C03652=1111.482,258.279,-73.038,-178.384,10.028,149.558
C03653=1111.486,258.031,-73.009,-178.387,10.025,149.558
C03654=1111.491,257.782,-72.980,-178.389,10.023,149.558
C03655=1111.494,257.534,-72.951,-178.392,10.020,149.558
C03656=1111.499,257.286,-72.923,-178.395,10.017,149.558
C03657=1111.503,257.038,-72.894,-178.398,10.014,149.558
C03658=1111.507,256.790,-72.864,-178.401,10.011,149.558
C03659=1111.511,256.541,-72.836,-178.404,10.009,149.558
C03660=1111.516,256.293,-72.807,-178.406,10.006,149.558
C03661=1111.520,256.045,-72.778,-178.409,10.003,149.558
C03662=1111.524,255.832,-72.754,-178.410,10.001,149.558
C03663=1111.527,255.619,-72.729,-178.412,9.999,149.558
C03664=1111.531,255.406,-72.704,-178.414,9.998,149.558
C03665=1111.535,255.194,-72.680,-178.416,9.995,149.558
C03666=1111.538,254.981,-72.655,-178.418,9.993,149.558
C03667=1111.542,254.768,-72.630,-178.419,9.992,149.558
C03668=1111.545,254.555,-72.606,-178.422,9.990,149.559
C03669=1111.550,254.343,-72.581,-178.424,9.988,149.559
C03670=1111.554,254.094,-72.552,-178.426,9.986,149.559
C03671=1111.558,253.846,-72.524,-178.429,9.983,149.559
C03672=1111.562,253.598,-72.495,-178.431,9.981,149.559
C03673=1111.567,253.349,-72.466,-178.433,9.979,149.559
C03674=1111.571,253.101,-72.438,-178.436,9.976,149.559
C03675=1111.575,252.853,-72.408,-178.439,9.974,149.559
C03676=1111.579,252.605,-72.380,-178.442,9.971,149.559
C03677=1111.584,252.356,-72.352,-178.445,9.969,149.559
C03678=1111.587,252.108,-72.323,-178.447,9.967,149.560
C03679=1111.592,251.860,-72.294,-178.450,9.964,149.560
C03680=1111.597,251.611,-72.266,-178.453,9.962,149.560
C03681=1111.600,251.363,-72.237,-178.457,9.959,149.560
C03682=1111.605,251.115,-72.209,-178.460,9.956,149.560
C03683=1111.609,250.866,-72.180,-178.462,9.954,149.561
C03684=1111.614,250.618,-72.152,-178.466,9.951,149.561
C03685=1111.617,250.370,-72.123,-178.469,9.948,149.561
C03686=1111.622,250.121,-72.094,-178.472,9.946,149.561
C03687=1111.626,249.873,-72.067,-178.475,9.943,149.561
C03688=1111.631,249.624,-72.038,-178.479,9.940,149.562
C03689=1111.634,249.376,-72.010,-178.482,9.937,149.562
C03690=1111.640,249.128,-71.981,-178.485,9.935,149.562
C03691=1111.643,248.880,-71.953,-178.489,9.931,149.562
C03692=1111.647,248.632,-71.925,-178.492,9.928,149.562
C03693=1111.652,248.383,-71.896,-178.495,9.925,149.562
C03694=1111.656,248.134,-71.868,-178.499,9.922,149.563
C03695=1111.661,247.886,-71.839,-178.503,9.918,149.563
C03696=1111.664,247.637,-71.811,-178.506,9.915,149.563
C03697=1111.670,247.389,-71.783,-178.509,9.911,149.563
C03698=1111.673,247.141,-71.755,-178.511,9.908,149.563
C03699=1111.678,246.893,-71.727,-178.514,9.906,149.563
C03700=1111.682,246.644,-71.698,-178.516,9.903,149.563
C03701=1111.686,246.396,-71.671,-178.518,9.901,149.563
C03702=1111.690,246.147,-71.642,-178.520,9.898,149.562
C03703=1111.695,245.899,-71.614,-178.523,9.895,149.562
C03704=1111.699,245.651,-71.586,-178.525,9.892,149.562
C03705=1111.703,245.402,-71.558,-178.528,9.890,149.562
C03706=1111.708,245.154,-71.529,-178.530,9.887,149.562
C03707=1111.712,244.905,-71.501,-178.532,9.884,149.562
C03708=1111.716,244.657,-71.473,-178.535,9.882,149.562
C03709=1111.720,244.409,-71.445,-178.537,9.879,149.562
C03710=1111.725,244.161,-71.417,-178.539,9.877,149.562
C03711=1111.729,243.912,-71.390,-178.542,9.874,149.562
C03712=1111.733,243.664,-71.362,-178.544,9.872,149.562
C03713=1111.738,243.415,-71.333,-178.547,9.869,149.562
C03714=1111.742,243.167,-71.305,-178.549,9.867,149.562
C03715=1111.746,242.919,-71.277,-178.552,9.864,149.563
C03716=1111.750,242.670,-71.249,-178.554,9.861,149.562
C03717=1111.756,242.422,-71.222,-178.556,9.859,149.563
C03718=1111.759,242.209,-71.197,-178.558,9.856,149.563
C03719=1111.762,241.996,-71.174,-178.561,9.854,149.563
C03720=1111.766,241.783,-71.149,-178.563,9.852,149.563
C03721=1111.769,241.570,-71.126,-178.565,9.850,149.563
C03722=1111.774,241.357,-71.102,-178.567,9.847,149.563
C03723=1111.777,241.144,-71.078,-178.570,9.845,149.563
C03724=1111.781,240.931,-71.054,-178.572,9.843,149.563
C03725=1111.785,240.718,-71.030,-178.574,9.841,149.563
C03726=1111.789,240.470,-71.003,-178.576,9.839,149.563
C03727=1111.793,240.222,-70.975,-178.579,9.836,149.563
C03728=1111.797,239.974,-70.947,-178.582,9.833,149.563
C03729=1111.802,239.724,-70.919,-178.584,9.831,149.563
C03730=1111.806,239.477,-70.891,-178.587,9.828,149.563
C03731=1111.811,239.228,-70.864,-178.589,9.826,149.563
C03732=1111.815,238.980,-70.836,-178.592,9.823,149.563
C03733=1111.819,238.732,-70.808,-178.595,9.820,149.564
C03734=1111.823,238.482,-70.781,-178.597,9.818,149.563
C03735=1111.827,238.235,-70.753,-178.600,9.815,149.564
C03736=1111.832,237.987,-70.725,-178.603,9.812,149.564
C03737=1111.836,237.738,-70.698,-178.605,9.811,149.564
C03738=1111.841,237.489,-70.669,-178.608,9.808,149.564
C03739=1111.846,237.241,-70.642,-178.610,9.805,149.564
C03740=1111.849,236.992,-70.614,-178.613,9.803,149.564
C03741=1111.854,236.744,-70.587,-178.616,9.800,149.564
C03742=1111.858,236.496,-70.559,-178.618,9.797,149.564
C03743=1111.862,236.247,-70.532,-178.621,9.794,149.564
C03744=1111.867,235.999,-70.504,-178.623,9.792,149.564
C03745=1111.871,235.750,-70.477,-178.626,9.789,149.564
C03746=1111.875,235.502,-70.449,-178.629,9.787,149.565
C03747=1111.880,235.253,-70.422,-178.632,9.784,149.565
C03748=1111.884,235.005,-70.395,-178.634,9.782,149.565
C03749=1111.888,234.756,-70.367,-178.637,9.779,149.565
C03750=1111.893,234.508,-70.339,-178.640,9.776,149.565
C03751=1111.897,234.260,-70.312,-178.643,9.773,149.565
C03752=1111.901,234.011,-70.284,-178.646,9.771,149.565
C03753=1111.906,233.762,-70.257,-178.648,9.767,149.565
C03754=1111.910,233.514,-70.229,-178.651,9.765,149.565
C03755=1111.915,233.266,-70.202,-178.654,9.763,149.565
C03756=1111.918,233.017,-70.176,-178.657,9.760,149.565
C03757=1111.923,232.769,-70.148,-178.660,9.757,149.566
C03758=1111.927,232.520,-70.121,-178.662,9.754,149.566
C03759=1111.932,232.272,-70.094,-178.665,9.751,149.566
C03760=1111.936,232.023,-70.065,-178.668,9.749,149.566
C03761=1111.940,231.775,-70.038,-178.670,9.745,149.566
C03762=1111.945,231.526,-70.011,-178.673,9.743,149.566
C03763=1111.950,231.278,-69.984,-178.676,9.740,149.566
C03764=1111.953,231.029,-69.956,-178.679,9.737,149.566
C03765=1111.957,230.781,-69.930,-178.682,9.734,149.566
C03766=1111.962,230.533,-69.903,-178.685,9.731,149.566
C03767=1111.967,230.284,-69.876,-178.687,9.728,149.566
C03768=1111.971,230.035,-69.848,-178.690,9.726,149.566
C03769=1111.975,229.786,-69.821,-178.693,9.723,149.566
C03770=1111.980,229.539,-69.793,-178.696,9.720,149.566
C03771=1111.984,229.290,-69.767,-178.699,9.717,149.566
C03772=1111.988,229.042,-69.740,-178.701,9.714,149.566
C03773=1111.993,228.793,-69.713,-178.704,9.711,149.566
C03774=1111.997,228.580,-69.689,-178.707,9.708,149.566
C03775=1112.001,228.367,-69.666,-178.709,9.706,149.566
C03776=1112.004,228.154,-69.644,-178.711,9.704,149.566
C03777=1112.007,227.941,-69.620,-178.713,9.701,149.566
C03778=1112.011,227.728,-69.596,-178.716,9.699,149.566
C03779=1112.015,227.514,-69.574,-178.718,9.695,149.566
C03780=1112.019,227.302,-69.551,-178.720,9.693,149.566
C03781=1112.022,227.089,-69.528,-178.723,9.690,149.566
C03782=1112.027,226.841,-69.501,-178.726,9.687,149.566
C03783=1112.032,226.592,-69.474,-178.728,9.684,149.566
C03784=1112.035,226.343,-69.447,-178.731,9.681,149.566
C03785=1112.040,226.095,-69.420,-178.733,9.678,149.566
C03786=1112.044,225.846,-69.393,-178.736,9.675,149.566
C03787=1112.048,225.598,-69.366,-178.739,9.672,149.566
C03788=1112.053,225.349,-69.340,-178.741,9.669,149.566
C03789=1112.058,225.101,-69.313,-178.744,9.666,149.566
C03790=1112.062,224.853,-69.286,-178.746,9.663,149.566
C03791=1112.067,224.604,-69.259,-178.749,9.660,149.566
C03792=1112.070,224.356,-69.233,-178.751,9.657,149.566
C03793=1112.075,224.107,-69.206,-178.754,9.653,149.566
C03794=1112.079,223.858,-69.178,-178.756,9.650,149.566
C03795=1112.083,223.609,-69.152,-178.759,9.647,149.566
C03796=1112.088,223.361,-69.125,-178.761,9.644,149.566
C03797=1112.092,223.113,-69.099,-178.764,9.641,149.566
C03798=1112.097,222.864,-69.072,-178.766,9.638,149.566
C03799=1112.101,222.616,-69.045,-178.769,9.635,149.565
C03800=1112.106,222.367,-69.019,-178.771,9.632,149.565
C03801=1112.110,222.118,-68.992,-178.774,9.629,149.565
C03802=1112.114,221.870,-68.966,-178.777,9.625,149.565
C03803=1112.119,221.621,-68.939,-178.778,9.623,149.565
C03804=1112.123,221.373,-68.913,-178.781,9.620,149.565
C03805=1112.128,221.124,-68.886,-178.783,9.617,149.565
C03806=1112.132,220.876,-68.860,-178.786,9.614,149.565
C03807=1112.137,220.627,-68.833,-178.788,9.610,149.565
C03808=1112.140,220.379,-68.806,-178.791,9.607,149.565
C03809=1112.145,220.130,-68.780,-178.793,9.604,149.565
C03810=1112.149,219.882,-68.754,-178.796,9.601,149.565
C03811=1112.154,219.633,-68.727,-178.798,9.598,149.564
C03812=1112.158,219.384,-68.701,-178.800,9.595,149.564
C03813=1112.163,219.136,-68.674,-178.802,9.592,149.564
C03814=1112.167,218.887,-68.648,-178.805,9.589,149.564
C03815=1112.171,218.639,-68.621,-178.807,9.586,149.564
C03816=1112.176,218.390,-68.594,-178.810,9.583,149.564
C03817=1112.180,218.142,-68.569,-178.812,9.580,149.564
C03818=1112.185,217.893,-68.542,-178.814,9.577,149.564
C03819=1112.189,217.644,-68.516,-178.816,9.574,149.564
C03820=1112.193,217.396,-68.489,-178.819,9.571,149.564
C03821=1112.198,217.147,-68.463,-178.821,9.568,149.563
C03822=1112.202,216.899,-68.437,-178.823,9.565,149.563
C03823=1112.206,216.651,-68.411,-178.825,9.562,149.563
C03824=1112.211,216.402,-68.385,-178.828,9.559,149.563
C03825=1112.215,216.153,-68.358,-178.830,9.556,149.563
C03826=1112.219,215.905,-68.333,-178.832,9.553,149.563
C03827=1112.224,215.656,-68.306,-178.834,9.550,149.563
C03828=1112.228,215.407,-68.280,-178.837,9.547,149.563
C03829=1112.232,215.159,-68.253,-178.839,9.544,149.563
C03830=1112.237,214.946,-68.231,-178.840,9.542,149.562
C03831=1112.240,214.733,-68.209,-178.843,9.538,149.562
C03832=1112.244,214.519,-68.186,-178.845,9.536,149.562
C03833=1112.248,214.307,-68.164,-178.847,9.534,149.562
C03834=1112.251,214.093,-68.142,-178.848,9.531,149.562
C03835=1112.256,213.880,-68.119,-178.850,9.529,149.562
C03836=1112.259,213.667,-68.097,-178.852,9.526,149.562
C03837=1112.263,213.454,-68.074,-178.854,9.524,149.562
C03838=1112.267,213.205,-68.048,-178.856,9.521,149.562
C03839=1112.272,212.956,-68.022,-178.860,9.517,149.562
C03840=1112.276,212.708,-67.997,-178.862,9.514,149.562
C03841=1112.281,212.460,-67.970,-178.865,9.511,149.562
C03842=1112.285,212.211,-67.944,-178.868,9.508,149.562
C03843=1112.290,211.962,-67.918,-178.871,9.505,149.562
C03844=1112.294,211.713,-67.893,-178.874,9.501,149.562
C03845=1112.298,211.465,-67.866,-178.876,9.499,149.562
C03846=1112.303,211.217,-67.840,-178.879,9.496,149.562
C03847=1112.307,210.968,-67.814,-178.882,9.493,149.562
C03848=1112.312,210.719,-67.789,-178.885,9.489,149.562
C03849=1112.316,210.470,-67.763,-178.888,9.486,149.562
C03850=1112.320,210.221,-67.737,-178.891,9.483,149.562
C03851=1112.325,209.973,-67.712,-178.894,9.480,149.562
C03852=1112.330,209.725,-67.685,-178.896,9.478,149.562
C03853=1112.334,209.476,-67.659,-178.899,9.475,149.562
C03854=1112.338,209.227,-67.633,-178.903,9.471,149.562
C03855=1112.343,208.979,-67.608,-178.905,9.468,149.562
C03856=1112.347,208.730,-67.582,-178.908,9.465,149.562
C03857=1112.351,208.482,-67.556,-178.911,9.462,149.563
C03858=1112.356,208.233,-67.531,-178.914,9.459,149.562
C03859=1112.360,207.985,-67.505,-178.916,9.457,149.563
C03860=1112.365,207.736,-67.479,-178.919,9.454,149.563
C03861=1112.369,207.487,-67.454,-178.922,9.451,149.563
C03862=1112.373,207.238,-67.428,-178.925,9.448,149.563
C03863=1112.378,206.990,-67.403,-178.928,9.445,149.563
C03864=1112.382,206.741,-67.377,-178.931,9.442,149.563
C03865=1112.386,206.492,-67.351,-178.934,9.439,149.563
C03866=1112.391,206.244,-67.326,-178.937,9.436,149.563
C03867=1112.396,205.995,-67.301,-178.940,9.433,149.563
C03868=1112.400,205.746,-67.275,-178.943,9.430,149.563
C03869=1112.405,205.498,-67.249,-178.945,9.427,149.563
C03870=1112.409,205.249,-67.224,-178.948,9.425,149.564
C03871=1112.413,205.000,-67.198,-178.951,9.422,149.564
C03872=1112.418,204.752,-67.173,-178.954,9.419,149.564
C03873=1112.423,204.503,-67.148,-178.957,9.416,149.564
C03874=1112.427,204.254,-67.122,-178.960,9.413,149.564
C03875=1112.432,204.006,-67.096,-178.963,9.410,149.564
C03876=1112.436,203.757,-67.071,-178.966,9.408,149.564
C03877=1112.441,203.508,-67.046,-178.968,9.405,149.564
C03878=1112.445,203.260,-67.020,-178.971,9.402,149.564
C03879=1112.449,203.011,-66.995,-178.974,9.399,149.564
C03880=1112.454,202.763,-66.969,-178.976,9.396,149.564
C03881=1112.459,202.513,-66.944,-178.980,9.392,149.565
C03882=1112.462,202.265,-66.919,-178.983,9.390,149.565
C03883=1112.467,202.017,-66.894,-178.986,9.387,149.565
C03884=1112.472,201.767,-66.869,-178.988,9.384,149.565
C03885=1112.476,201.519,-66.843,-178.991,9.381,149.565
C03886=1112.480,201.305,-66.822,-178.993,9.379,149.565
C03887=1112.484,201.093,-66.800,-178.996,9.376,149.565
C03888=1112.488,200.879,-66.778,-178.998,9.374,149.565
C03889=1112.491,200.666,-66.757,-179.001,9.371,149.565
C03890=1112.496,200.453,-66.735,-179.003,9.369,149.565
C03891=1112.499,200.239,-66.713,-179.006,9.366,149.565
C03892=1112.503,200.026,-66.692,-179.008,9.364,149.565
C03893=1112.506,199.813,-66.670,-179.011,9.361,149.565
C03894=1112.512,199.564,-66.645,-179.013,9.358,149.565
C03895=1112.515,199.316,-66.620,-179.016,9.355,149.565
C03896=1112.520,199.067,-66.595,-179.019,9.352,149.565
C03897=1112.524,198.818,-66.570,-179.021,9.349,149.565
C03898=1112.530,198.569,-66.545,-179.024,9.346,149.565
C03899=1112.533,198.321,-66.520,-179.027,9.343,149.565
C03900=1112.538,198.072,-66.495,-179.029,9.340,149.565
C03901=1112.542,197.823,-66.469,-179.033,9.336,149.565
C03902=1112.547,197.575,-66.445,-179.035,9.333,149.565
C03903=1112.551,197.326,-66.420,-179.038,9.330,149.565
C03904=1112.556,197.077,-66.395,-179.041,9.327,149.565
C03905=1112.560,196.828,-66.370,-179.043,9.324,149.565
C03906=1112.565,196.580,-66.345,-179.046,9.321,149.565
C03907=1112.569,196.331,-66.320,-179.049,9.318,149.565
C03908=1112.574,196.082,-66.296,-179.051,9.315,149.565
C03909=1112.578,195.834,-66.270,-179.052,9.312,149.565
C03910=1112.582,195.585,-66.246,-179.055,9.309,149.565
C03911=1112.587,195.336,-66.221,-179.056,9.306,149.565
C03912=1112.592,195.087,-66.196,-179.059,9.303,149.565
C03913=1112.596,194.839,-66.172,-179.061,9.301,149.565
C03914=1112.601,194.590,-66.147,-179.063,9.297,149.564
C03915=1112.605,194.341,-66.123,-179.065,9.295,149.564
C03916=1112.609,194.093,-66.097,-179.067,9.292,149.564
C03917=1112.614,193.844,-66.072,-179.069,9.290,149.564
C03918=1112.619,193.595,-66.048,-179.071,9.287,149.564
C03919=1112.623,193.346,-66.023,-179.073,9.284,149.564
C03920=1112.627,193.098,-65.998,-179.075,9.282,149.564
C03921=1112.632,192.849,-65.973,-179.078,9.278,149.564
C03922=1112.636,192.600,-65.949,-179.080,9.276,149.564
C03923=1112.641,192.352,-65.924,-179.082,9.273,149.564
C03924=1112.645,192.103,-65.900,-179.085,9.270,149.564
C03925=1112.650,191.854,-65.875,-179.087,9.268,149.564
C03926=1112.654,191.605,-65.850,-179.089,9.264,149.563
C03927=1112.659,191.357,-65.826,-179.091,9.262,149.563
C03928=1112.663,191.108,-65.801,-179.093,9.259,149.563
C03929=1112.668,190.859,-65.776,-179.095,9.256,149.563
C03930=1112.672,190.610,-65.752,-179.097,9.253,149.563
C03931=1112.677,190.362,-65.728,-179.099,9.251,149.563
C03932=1112.681,190.113,-65.703,-179.102,9.248,149.563
C03933=1112.686,189.864,-65.679,-179.104,9.245,149.563
C03934=1112.691,189.615,-65.654,-179.106,9.242,149.563
C03935=1112.695,189.366,-65.629,-179.109,9.239,149.563
C03936=1112.700,189.118,-65.605,-179.111,9.237,149.563
C03937=1112.705,188.869,-65.581,-179.113,9.234,149.563
C03938=1112.709,188.620,-65.556,-179.115,9.231,149.563
C03939=1112.713,188.371,-65.532,-179.118,9.228,149.563
C03940=1112.718,188.123,-65.508,-179.120,9.225,149.563
C03941=1112.722,187.873,-65.483,-179.122,9.223,149.563
C03942=1112.726,187.660,-65.462,-179.124,9.221,149.563
C03943=1112.730,187.447,-65.441,-179.126,9.217,149.563
C03944=1112.734,187.234,-65.420,-179.128,9.215,149.563
C03945=1112.738,187.021,-65.399,-179.130,9.213,149.563
C03946=1112.742,186.807,-65.378,-179.132,9.210,149.563
C03947=1112.745,186.593,-65.358,-179.134,9.208,149.563
C03948=1112.750,186.380,-65.337,-179.136,9.206,149.563
C03949=1112.753,186.167,-65.316,-179.138,9.203,149.563
C03950=1112.758,185.918,-65.292,-179.140,9.200,149.562
C03951=1112.762,185.669,-65.267,-179.143,9.198,149.563
C03952=1112.766,185.421,-65.243,-179.146,9.194,149.563
C03953=1112.772,185.172,-65.218,-179.148,9.192,149.563
C03954=1112.776,184.923,-65.195,-179.150,9.189,149.563
C03955=1112.780,184.674,-65.171,-179.153,9.186,149.562
C03956=1112.785,184.425,-65.146,-179.155,9.184,149.562
C03957=1112.790,184.177,-65.122,-179.157,9.180,149.562
C03958=1112.794,183.928,-65.098,-179.160,9.177,149.562
C03959=1112.799,183.679,-65.074,-179.162,9.174,149.562
C03960=1112.803,183.430,-65.049,-179.165,9.171,149.562
C03961=1112.808,183.182,-65.025,-179.167,9.169,149.562
C03962=1112.812,182.933,-65.001,-179.169,9.166,149.562
C03963=1112.817,182.684,-64.978,-179.172,9.163,149.562
C03964=1112.820,182.435,-64.953,-179.174,9.160,149.562
C03965=1112.826,182.186,-64.929,-179.177,9.156,149.562
C03966=1112.830,181.937,-64.905,-179.179,9.153,149.562
C03967=1112.835,181.689,-64.881,-179.181,9.151,149.562
C03968=1112.839,181.440,-64.857,-179.184,9.148,149.562
C03969=1112.844,181.191,-64.834,-179.186,9.145,149.562
C03970=1112.848,180.942,-64.809,-179.189,9.142,149.562
C03971=1112.853,180.694,-64.785,-179.191,9.139,149.562
C03972=1112.857,180.445,-64.761,-179.194,9.135,149.562
C03973=1112.862,180.196,-64.737,-179.196,9.132,149.562
C03974=1112.866,179.947,-64.714,-179.199,9.129,149.562
C03975=1112.871,179.699,-64.690,-179.201,9.126,149.562
C03976=1112.876,179.450,-64.667,-179.204,9.123,149.562
C03977=1112.879,179.201,-64.642,-179.206,9.119,149.561
C03978=1112.884,178.952,-64.618,-179.208,9.117,149.561
C03979=1112.889,178.703,-64.594,-179.210,9.114,149.561
C03980=1112.894,178.454,-64.570,-179.212,9.111,149.561
C03981=1112.898,178.205,-64.547,-179.214,9.108,149.561
C03982=1112.903,177.957,-64.523,-179.217,9.105,149.561
C03983=1112.907,177.708,-64.499,-179.219,9.102,149.561
C03984=1112.912,177.459,-64.476,-179.221,9.099,149.561
C03985=1112.916,177.210,-64.452,-179.223,9.096,149.561
C03986=1112.921,176.961,-64.428,-179.225,9.093,149.560
C03987=1112.925,176.712,-64.404,-179.227,9.090,149.560
C03988=1112.930,176.463,-64.381,-179.230,9.087,149.560
C03989=1112.934,176.215,-64.357,-179.231,9.085,149.560
C03990=1112.939,175.966,-64.333,-179.234,9.081,149.560
C03991=1112.943,175.717,-64.310,-179.236,9.078,149.560
C03992=1112.948,175.468,-64.286,-179.238,9.076,149.560
C03993=1112.953,175.219,-64.262,-179.240,9.073,149.560
C03994=1112.957,174.970,-64.239,-179.243,9.069,149.560
C03995=1112.962,174.722,-64.215,-179.244,9.067,149.559
C03996=1112.966,174.473,-64.192,-179.247,9.064,149.559
C03997=1112.971,174.224,-64.168,-179.249,9.061,149.559
C03998=1112.975,174.011,-64.148,-179.251,9.058,149.559
C03999=1112.978,173.797,-64.128,-179.253,9.055,149.559
C04000=1112.983,173.583,-64.108,-179.255,9.053,149.559
C04001=1112.987,173.370,-64.088,-179.257,9.051,149.559
C04002=1112.990,173.157,-64.067,-179.259,9.047,149.559
C04003=1112.994,172.943,-64.047,-179.261,9.045,149.559
C04004=1112.998,172.730,-64.027,-179.262,9.043,149.559
C04005=1113.002,172.516,-64.007,-179.264,9.040,149.559
C04006=1113.007,172.268,-63.983,-179.266,9.037,149.558
C04007=1113.011,172.019,-63.960,-179.268,9.035,149.558
C04008=1113.016,171.770,-63.936,-179.271,9.031,149.558
C04009=1113.020,171.521,-63.914,-179.273,9.028,149.558
C04010=1113.025,171.272,-63.890,-179.275,9.026,149.558
C04011=1113.029,171.023,-63.866,-179.277,9.022,149.558
C04012=1113.034,170.774,-63.843,-179.279,9.019,149.558
C04013=1113.038,170.525,-63.820,-179.282,9.016,149.558
C04014=1113.043,170.276,-63.796,-179.284,9.014,149.558
C04015=1113.048,170.027,-63.773,-179.286,9.010,149.557
C04016=1113.052,169.778,-63.750,-179.288,9.007,149.557
C04017=1113.057,169.530,-63.727,-179.290,9.005,149.557
C04018=1113.062,169.281,-63.704,-179.292,9.001,149.557
C04019=1113.066,169.032,-63.680,-179.295,8.998,149.557
C04020=1113.071,168.783,-63.657,-179.297,8.995,149.557
C04021=1113.075,168.534,-63.634,-179.299,8.992,149.557
C04022=1113.080,168.285,-63.611,-179.301,8.989,149.557
C04023=1113.084,168.036,-63.588,-179.304,8.986,149.557
C04024=1113.089,167.787,-63.564,-179.305,8.983,149.557
C04025=1113.093,167.539,-63.541,-179.308,8.980,149.556
C04026=1113.098,167.289,-63.518,-179.310,8.977,149.556
C04027=1113.103,167.041,-63.495,-179.313,8.974,149.556
C04028=1113.108,166.792,-63.472,-179.314,8.971,149.556
C04029=1113.112,166.543,-63.449,-179.317,8.968,149.556
C04030=1113.117,166.294,-63.426,-179.319,8.965,149.556
C04031=1113.121,166.045,-63.402,-179.322,8.962,149.556
C04032=1113.125,165.797,-63.379,-179.323,8.959,149.556
C04033=1113.130,165.548,-63.356,-179.326,8.956,149.556
C04034=1113.135,165.299,-63.333,-179.328,8.952,149.555
C04035=1113.139,165.051,-63.310,-179.330,8.949,149.555
C04036=1113.144,164.802,-63.287,-179.333,8.946,149.555
C04037=1113.149,164.552,-63.264,-179.334,8.943,149.555
C04038=1113.153,164.303,-63.242,-179.337,8.940,149.555
C04039=1113.158,164.054,-63.218,-179.339,8.937,149.555
C04040=1113.163,163.806,-63.195,-179.341,8.934,149.555
C04041=1113.167,163.557,-63.172,-179.343,8.931,149.555
C04042=1113.172,163.307,-63.150,-179.345,8.928,149.554
C04043=1113.176,163.059,-63.127,-179.348,8.925,149.554
C04044=1113.180,162.810,-63.104,-179.350,8.921,149.554
C04045=1113.185,162.562,-63.081,-179.352,8.918,149.554
C04046=1113.190,162.312,-63.059,-179.354,8.915,149.554
C04047=1113.195,162.063,-63.035,-179.356,8.912,149.554
C04048=1113.199,161.814,-63.013,-179.358,8.909,149.554
C04049=1113.203,161.565,-62.989,-179.361,8.906,149.554
C04050=1113.208,161.317,-62.967,-179.363,8.902,149.553
C04051=1113.213,161.068,-62.944,-179.366,8.899,149.553
C04052=1113.217,160.819,-62.921,-179.367,8.896,149.553
C04053=1113.222,160.569,-62.899,-179.370,8.893,149.553
C04054=1113.226,160.356,-62.879,-179.372,8.890,149.553
C04055=1113.230,160.143,-62.859,-179.373,8.887,149.553
C04056=1113.234,159.929,-62.840,-179.375,8.885,149.553
C04057=1113.237,159.715,-62.821,-179.377,8.882,149.553
C04058=1113.241,159.502,-62.801,-179.379,8.879,149.553
C04059=1113.246,159.288,-62.783,-179.381,8.877,149.552
C04060=1113.249,159.075,-62.763,-179.383,8.874,149.552
C04061=1113.253,158.861,-62.743,-179.385,8.871,149.552
C04062=1113.258,158.611,-62.720,-179.387,8.868,149.552
C04063=1113.263,158.363,-62.698,-179.389,8.864,149.552
C04064=1113.267,158.114,-62.676,-179.391,8.861,149.552
C04065=1113.272,157.865,-62.653,-179.393,8.858,149.551
C04066=1113.277,157.616,-62.631,-179.395,8.855,149.551
C04067=1113.281,157.367,-62.608,-179.398,8.852,149.551
C04068=1113.286,157.118,-62.586,-179.400,8.848,149.551
C04069=1113.290,156.870,-62.563,-179.402,8.845,149.551
C04070=1113.295,156.620,-62.540,-179.405,8.842,149.551
C04071=1113.299,156.372,-62.518,-179.407,8.838,149.550
C04072=1113.305,156.123,-62.495,-179.409,8.835,149.550
C04073=1113.309,155.874,-62.473,-179.411,8.832,149.550
C04074=1113.313,155.625,-62.451,-179.413,8.828,149.550
C04075=1113.319,155.376,-62.428,-179.415,8.825,149.550
C04076=1113.323,155.127,-62.406,-179.417,8.822,149.550
C04077=1113.327,154.878,-62.384,-179.419,8.819,149.549
C04078=1113.332,154.629,-62.361,-179.422,8.815,149.549
C04079=1113.336,154.380,-62.339,-179.424,8.812,149.549
C04080=1113.341,154.131,-62.317,-179.426,8.809,149.549
C04081=1113.346,153.882,-62.293,-179.428,8.805,149.549
C04082=1113.350,153.633,-62.271,-179.430,8.802,149.548
C04083=1113.355,153.384,-62.250,-179.433,8.799,149.548
C04084=1113.359,153.135,-62.228,-179.435,8.795,149.548
C04085=1113.365,152.887,-62.205,-179.437,8.792,149.548
C04086=1113.369,152.637,-62.183,-179.439,8.788,149.548
C04087=1113.373,152.388,-62.161,-179.441,8.785,149.547
C04088=1113.378,152.139,-62.139,-179.444,8.782,149.547
C04089=1113.383,151.890,-62.116,-179.446,8.778,149.547
C04090=1113.388,151.642,-62.094,-179.448,8.775,149.547
C04091=1113.392,151.392,-62.072,-179.450,8.771,149.547
C04092=1113.397,151.144,-62.050,-179.452,8.768,149.546
C04093=1113.402,150.894,-62.027,-179.454,8.764,149.546
C04094=1113.406,150.646,-62.005,-179.456,8.761,149.546
C04095=1113.411,150.397,-61.983,-179.458,8.757,149.546
C04096=1113.415,150.148,-61.961,-179.461,8.753,149.546
C04097=1113.420,149.899,-61.939,-179.463,8.750,149.546
C04098=1113.425,149.650,-61.918,-179.466,8.746,149.545
C04099=1113.430,149.400,-61.895,-179.468,8.743,149.545
C04100=1113.434,149.152,-61.873,-179.470,8.739,149.545
C04101=1113.439,148.902,-61.851,-179.472,8.736,149.545
C04102=1113.444,148.654,-61.830,-179.474,8.732,149.544
C04103=1113.448,148.404,-61.808,-179.476,8.729,149.544
C04104=1113.453,148.156,-61.786,-179.478,8.725,149.544
C04105=1113.457,147.906,-61.764,-179.480,8.722,149.544
C04106=1113.462,147.658,-61.741,-179.482,8.718,149.543
C04107=1113.467,147.409,-61.719,-179.485,8.714,149.543
C04108=1113.472,147.160,-61.698,-179.487,8.711,149.543
C04109=1113.476,146.910,-61.676,-179.489,8.707,149.542
C04110=1113.480,146.698,-61.657,-179.490,8.704,149.542
C04111=1113.484,146.483,-61.638,-179.493,8.701,149.542
C04112=1113.488,146.270,-61.620,-179.495,8.697,149.542
C04113=1113.492,146.056,-61.601,-179.496,8.695,149.542
C04114=1113.496,145.842,-61.582,-179.498,8.691,149.542
C04115=1113.500,145.629,-61.563,-179.500,8.689,149.541
C04116=1113.504,145.415,-61.544,-179.502,8.685,149.541
C04117=1113.508,145.201,-61.526,-179.504,8.682,149.541
C04118=1113.512,144.952,-61.504,-179.505,8.678,149.540
C04119=1113.517,144.703,-61.482,-179.506,8.675,149.540
C04120=1113.522,144.455,-61.461,-179.509,8.671,149.540
C04121=1113.526,144.205,-61.439,-179.510,8.668,149.539
C04122=1113.531,143.956,-61.418,-179.512,8.665,149.539
C04123=1113.536,143.707,-61.396,-179.513,8.661,149.539
C04124=1113.540,143.458,-61.374,-179.515,8.658,149.538
C04125=1113.545,143.210,-61.352,-179.516,8.654,149.538
C04126=1113.550,142.960,-61.330,-179.518,8.651,149.538
C04127=1113.555,142.711,-61.309,-179.519,8.648,149.537
C04128=1113.559,142.462,-61.287,-179.522,8.644,149.537
C04129=1113.564,142.213,-61.266,-179.523,8.641,149.537
C04130=1113.568,141.965,-61.245,-179.525,8.637,149.536
C04131=1113.573,141.715,-61.223,-179.527,8.634,149.536
C04132=1113.577,141.466,-61.201,-179.528,8.631,149.536
C04133=1113.582,141.217,-61.180,-179.530,8.627,149.535
C04134=1113.587,140.967,-61.158,-179.531,8.624,149.535
C04135=1113.592,140.719,-61.137,-179.533,8.621,149.535
C04136=1113.597,140.470,-61.115,-179.535,8.617,149.534
C04137=1113.601,140.221,-61.093,-179.537,8.613,149.534
C04138=1113.605,139.972,-61.073,-179.538,8.611,149.534
C04139=1113.610,139.723,-61.051,-179.540,8.607,149.533
C04140=1113.615,139.473,-61.030,-179.542,8.603,149.533
C04141=1113.620,139.225,-61.008,-179.543,8.600,149.533
C04142=1113.624,138.976,-60.986,-179.545,8.597,149.533
C04143=1113.629,138.726,-60.965,-179.547,8.593,149.532
C04144=1113.633,138.478,-60.944,-179.548,8.590,149.532
C04145=1113.638,138.228,-60.923,-179.550,8.587,149.532
C04146=1113.643,137.979,-60.901,-179.552,8.583,149.531
C04147=1113.647,137.730,-60.879,-179.553,8.580,149.531
C04148=1113.652,137.482,-60.859,-179.555,8.577,149.531
C04149=1113.657,137.233,-60.837,-179.557,8.573,149.530
C04150=1113.661,136.983,-60.816,-179.558,8.570,149.530
C04151=1113.666,136.734,-60.794,-179.560,8.567,149.530
C04152=1113.671,136.485,-60.774,-179.562,8.563,149.529
C04153=1113.676,136.237,-60.752,-179.563,8.560,149.529
C04154=1113.680,135.987,-60.731,-179.565,8.556,149.529
C04155=1113.685,135.738,-60.709,-179.567,8.553,149.529
C04156=1113.689,135.489,-60.689,-179.569,8.550,149.528
C04157=1113.694,135.241,-60.667,-179.571,8.546,149.528
C04158=1113.699,134.991,-60.646,-179.572,8.543,149.528
C04159=1113.704,134.741,-60.625,-179.574,8.540,149.527
C04160=1113.708,134.493,-60.604,-179.576,8.536,149.527
C04161=1113.713,134.244,-60.583,-179.577,8.533,149.527
C04162=1113.718,133.995,-60.561,-179.579,8.530,149.526
C04163=1113.722,133.745,-60.540,-179.581,8.526,149.526
C04164=1113.727,133.496,-60.519,-179.582,8.524,149.526
C04165=1113.732,133.248,-60.498,-179.584,8.520,149.526
C04166=1113.736,133.034,-60.480,-179.585,8.517,149.525
C04167=1113.740,132.820,-60.462,-179.587,8.514,149.525
C04168=1113.744,132.606,-60.444,-179.589,8.511,149.525
C04169=1113.747,132.392,-60.426,-179.590,8.508,149.525
C04170=1113.752,132.179,-60.407,-179.592,8.505,149.524
C04171=1113.756,131.965,-60.390,-179.593,8.503,149.524
C04172=1113.760,131.751,-60.371,-179.595,8.500,149.524
C04173=1113.764,131.537,-60.354,-179.596,8.497,149.524
C04174=1113.769,131.288,-60.333,-179.598,8.493,149.523
C04175=1113.774,131.039,-60.311,-179.600,8.490,149.523
C04176=1113.778,130.790,-60.291,-179.601,8.487,149.523
C04177=1113.783,130.540,-60.269,-179.603,8.483,149.522
C04178=1113.787,130.292,-60.249,-179.605,8.480,149.522
C04179=1113.792,130.043,-60.227,-179.606,8.477,149.522
C04180=1113.797,129.794,-60.207,-179.608,8.474,149.522
C04181=1113.802,129.545,-60.186,-179.610,8.470,149.521
C04182=1113.807,129.295,-60.165,-179.612,8.467,149.521
C04183=1113.811,129.046,-60.145,-179.614,8.463,149.521
C04184=1113.816,128.798,-60.123,-179.616,8.460,149.521
C04185=1113.821,128.549,-60.103,-179.617,8.457,149.520
C04186=1113.825,128.299,-60.081,-179.619,8.453,149.520
C04187=1113.830,128.050,-60.061,-179.621,8.450,149.520
C04188=1113.835,127.801,-60.040,-179.622,8.447,149.520
C04189=1113.839,127.552,-60.020,-179.624,8.443,149.519
C04190=1113.845,127.302,-59.999,-179.626,8.440,149.519
C04191=1113.849,127.054,-59.978,-179.627,8.437,149.519
C04192=1113.854,126.804,-59.957,-179.629,8.434,149.518
C04193=1113.858,126.556,-59.936,-179.631,8.430,149.518
C04194=1113.863,126.307,-59.916,-179.633,8.427,149.518
C04195=1113.868,126.058,-59.895,-179.635,8.423,149.518
C04196=1113.872,125.809,-59.874,-179.637,8.420,149.517
C04197=1113.877,125.560,-59.853,-179.638,8.417,149.517
C04198=1113.882,125.311,-59.833,-179.640,8.413,149.517
C04199=1113.886,125.061,-59.812,-179.642,8.410,149.516
C04200=1113.891,124.812,-59.791,-179.643,8.407,149.516
C04201=1113.895,124.563,-59.771,-179.645,8.403,149.516
C04202=1113.901,124.313,-59.750,-179.647,8.400,149.515
C04203=1113.905,124.065,-59.730,-179.649,8.396,149.515
C04204=1113.909,123.816,-59.709,-179.650,8.394,149.515
C04205=1113.915,123.566,-59.688,-179.652,8.390,149.515
C04206=1113.919,123.317,-59.669,-179.654,8.386,149.514
C04207=1113.924,123.068,-59.648,-179.656,8.383,149.514
C04208=1113.929,122.819,-59.627,-179.658,8.380,149.514
C04209=1113.933,122.570,-59.607,-179.660,8.376,149.514
C04210=1113.938,122.321,-59.587,-179.661,8.373,149.513
C04211=1113.943,122.071,-59.566,-179.663,8.370,149.513
C04212=1113.947,121.822,-59.545,-179.665,8.366,149.513
C04213=1113.952,121.573,-59.525,-179.667,8.363,149.513
C04214=1113.957,121.324,-59.505,-179.668,8.360,149.512
C04215=1113.962,121.075,-59.484,-179.670,8.356,149.512
C04216=1113.966,120.826,-59.464,-179.672,8.353,149.512
C04217=1113.972,120.577,-59.443,-179.673,8.350,149.511
C04218=1113.976,120.328,-59.423,-179.675,8.346,149.511
C04219=1113.981,120.079,-59.403,-179.677,8.343,149.511
C04220=1113.986,119.830,-59.383,-179.679,8.339,149.511
C04221=1113.991,119.580,-59.362,-179.681,8.336,149.510
C04222=1113.994,119.367,-59.345,-179.682,8.334,149.510
C04223=1113.998,119.152,-59.327,-179.684,8.330,149.510
C04224=1114.002,118.939,-59.310,-179.685,8.327,149.509
C04225=1114.006,118.725,-59.293,-179.687,8.324,149.509
C04226=1114.011,118.511,-59.275,-179.688,8.322,149.509
C04227=1114.015,118.297,-59.258,-179.689,8.319,149.509
C04228=1114.019,118.084,-59.240,-179.691,8.316,149.509
C04229=1114.023,117.869,-59.223,-179.693,8.313,149.508
C04230=1114.027,117.620,-59.202,-179.695,8.309,149.508
C04231=1114.033,117.371,-59.183,-179.696,8.307,149.508
C04232=1114.037,117.122,-59.162,-179.698,8.303,149.507
C04233=1114.042,116.873,-59.142,-179.700,8.299,149.507
C04234=1114.046,116.624,-59.122,-179.702,8.296,149.507
C04235=1114.051,116.374,-59.102,-179.703,8.293,149.507
C04236=1114.056,116.125,-59.082,-179.705,8.289,149.506
C04237=1114.061,115.876,-59.061,-179.707,8.286,149.506
C04238=1114.065,115.627,-59.041,-179.709,8.282,149.506
C04239=1114.070,115.378,-59.022,-179.710,8.279,149.505
C04240=1114.075,115.129,-59.001,-179.712,8.276,149.505
C04241=1114.080,114.880,-58.982,-179.714,8.272,149.505
C04242=1114.085,114.630,-58.961,-179.716,8.268,149.505
C04243=1114.089,114.381,-58.941,-179.718,8.265,149.504
C04244=1114.094,114.132,-58.921,-179.720,8.262,149.504
C04245=1114.099,113.883,-58.901,-179.722,8.258,149.504
C04246=1114.104,113.634,-58.881,-179.723,8.255,149.503
C04247=1114.108,113.384,-58.861,-179.725,8.251,149.503
C04248=1114.113,113.136,-58.841,-179.727,8.248,149.503
C04249=1114.118,112.886,-58.821,-179.728,8.244,149.503
C04250=1114.123,112.638,-58.801,-179.730,8.241,149.502
C04251=1114.127,112.388,-58.782,-179.732,8.237,149.502
C04252=1114.132,112.139,-58.761,-179.734,8.234,149.502
C04253=1114.137,111.890,-58.742,-179.736,8.231,149.501
C04254=1114.142,111.641,-58.722,-179.738,8.227,149.501
C04255=1114.146,111.392,-58.702,-179.739,8.223,149.501
C04256=1114.151,111.142,-58.682,-179.741,8.220,149.501
C04257=1114.156,110.893,-58.663,-179.743,8.216,149.500
C04258=1114.161,110.644,-58.643,-179.745,8.213,149.500
C04259=1114.166,110.395,-58.623,-179.747,8.209,149.500
C04260=1114.170,110.146,-58.603,-179.749,8.206,149.499
C04261=1114.175,109.896,-58.583,-179.751,8.202,149.499
C04262=1114.180,109.647,-58.564,-179.754,8.198,149.499
C04263=1114.185,109.398,-58.544,-179.756,8.194,149.499
C04264=1114.189,109.149,-58.524,-179.758,8.191,149.499
C04265=1114.194,108.899,-58.504,-179.760,8.187,149.498
C04266=1114.199,108.651,-58.485,-179.762,8.183,149.498
C04267=1114.204,108.401,-58.465,-179.764,8.180,149.498
C04268=1114.208,108.152,-58.445,-179.766,8.176,149.497
C04269=1114.213,107.903,-58.426,-179.768,8.172,149.497
C04270=1114.218,107.654,-58.406,-179.770,8.168,149.497
C04271=1114.223,107.404,-58.387,-179.772,8.165,149.497
C04272=1114.227,107.155,-58.366,-179.774,8.161,149.496
C04273=1114.232,106.906,-58.347,-179.776,8.157,149.496
C04274=1114.237,106.657,-58.327,-179.777,8.153,149.495
C04275=1114.241,106.408,-58.308,-179.779,8.150,149.495
C04276=1114.247,106.159,-58.289,-179.782,8.146,149.495
C04277=1114.251,105.909,-58.269,-179.784,8.142,149.495
C04278=1114.256,105.695,-58.252,-179.785,8.139,149.494
C04279=1114.259,105.481,-58.236,-179.787,8.136,149.494
C04280=1114.264,105.268,-58.219,-179.788,8.132,149.494
C04281=1114.267,105.053,-58.202,-179.790,8.129,149.494
C04282=1114.272,104.839,-58.186,-179.792,8.126,149.493
C04283=1114.276,104.626,-58.169,-179.793,8.122,149.493
C04284=1114.280,104.411,-58.152,-179.795,8.120,149.493
C04285=1114.284,104.198,-58.135,-179.797,8.116,149.492
C04286=1114.289,103.949,-58.116,-179.798,8.112,149.492
C04287=1114.294,103.699,-58.096,-179.800,8.109,149.492
C04288=1114.299,103.450,-58.077,-179.802,8.105,149.491
C04289=1114.303,103.201,-58.058,-179.804,8.101,149.491
C04290=1114.308,102.952,-58.038,-179.806,8.097,149.491
C04291=1114.313,102.703,-58.019,-179.807,8.094,149.490
C04292=1114.317,102.453,-58.001,-179.809,8.090,149.490
C04293=1114.323,102.204,-57.982,-179.811,8.086,149.490
C04294=1114.328,101.954,-57.962,-179.812,8.082,149.489
C04295=1114.332,101.706,-57.943,-179.815,8.079,149.489
C04296=1114.337,101.456,-57.924,-179.816,8.075,149.488
C04297=1114.342,101.207,-57.904,-179.818,8.071,149.488
C04298=1114.346,100.958,-57.885,-179.819,8.067,149.488
C04299=1114.351,100.709,-57.866,-179.821,8.064,149.487
C04300=1114.356,100.460,-57.846,-179.823,8.060,149.487
C04301=1114.360,100.210,-57.827,-179.825,8.056,149.487
C04302=1114.366,99.961,-57.809,-179.826,8.052,149.486
C04303=1114.371,99.711,-57.789,-179.828,8.048,149.486
C04304=1114.375,99.463,-57.770,-179.830,8.045,149.485
C04305=1114.380,99.213,-57.751,-179.831,8.041,149.485
C04306=1114.385,98.965,-57.732,-179.833,8.037,149.485
C04307=1114.390,98.714,-57.713,-179.835,8.033,149.484
C04308=1114.395,98.466,-57.694,-179.836,8.029,149.484
C04309=1114.399,98.216,-57.675,-179.838,8.025,149.483
C04310=1114.404,97.968,-57.655,-179.840,8.022,149.483
C04311=1114.409,97.718,-57.637,-179.842,8.018,149.483
C04312=1114.414,97.469,-57.618,-179.843,8.014,149.482
C04313=1114.418,97.220,-57.599,-179.845,8.010,149.482
C04314=1114.423,96.971,-57.579,-179.846,8.006,149.481
C04315=1114.428,96.721,-57.561,-179.848,8.002,149.481
C04316=1114.433,96.472,-57.542,-179.850,7.998,149.480
C04317=1114.437,96.223,-57.523,-179.851,7.994,149.480
C04318=1114.443,95.973,-57.504,-179.853,7.991,149.480
C04319=1114.447,95.725,-57.485,-179.854,7.987,149.479
C04320=1114.452,95.474,-57.466,-179.856,7.983,149.479
C04321=1114.457,95.226,-57.448,-179.858,7.979,149.478
C04322=1114.462,94.976,-57.428,-179.859,7.975,149.478
C04323=1114.467,94.727,-57.410,-179.860,7.972,149.477
C04324=1114.471,94.478,-57.390,-179.862,7.968,149.477
C04325=1114.476,94.228,-57.372,-179.863,7.964,149.477
C04326=1114.482,93.979,-57.353,-179.865,7.960,149.476
C04327=1114.486,93.730,-57.334,-179.867,7.956,149.476
C04328=1114.491,93.481,-57.316,-179.868,7.952,149.475
C04329=1114.495,93.231,-57.296,-179.869,7.948,149.475
C04330=1114.500,92.982,-57.278,-179.871,7.944,149.474
C04331=1114.506,92.733,-57.259,-179.872,7.941,149.474
C04332=1114.510,92.484,-57.241,-179.873,7.937,149.473
C04333=1114.514,92.235,-57.222,-179.875,7.933,149.473
C04334=1114.519,92.021,-57.205,-179.876,7.930,149.472
C04335=1114.523,91.806,-57.190,-179.878,7.926,149.472
C04336=1114.528,91.592,-57.174,-179.879,7.923,149.472
C04337=1114.531,91.378,-57.158,-179.880,7.920,149.471
C04338=1114.535,91.164,-57.142,-179.882,7.917,149.471
C04339=1114.540,90.950,-57.125,-179.883,7.914,149.470
C04340=1114.544,90.736,-57.110,-179.884,7.910,149.470
C04341=1114.548,90.522,-57.094,-179.884,7.907,149.470
C04342=1114.553,90.273,-57.076,-179.886,7.903,149.469
C04343=1114.558,90.023,-57.057,-179.887,7.899,149.469
C04344=1114.563,89.774,-57.038,-179.889,7.895,149.468
C04345=1114.567,89.525,-57.020,-179.890,7.891,149.468
C04346=1114.572,89.275,-57.002,-179.891,7.888,149.467
C04347=1114.577,89.027,-56.982,-179.893,7.884,149.467
C04348=1114.582,88.777,-56.964,-179.894,7.880,149.466
C04349=1114.586,88.527,-56.946,-179.896,7.876,149.466
C04350=1114.592,88.279,-56.927,-179.896,7.873,149.465
C04351=1114.597,88.029,-56.909,-179.898,7.869,149.465
C04352=1114.601,87.780,-56.890,-179.899,7.865,149.464
C04353=1114.606,87.531,-56.872,-179.901,7.861,149.464
C04354=1114.611,87.282,-56.853,-179.902,7.858,149.463
C04355=1114.616,87.032,-56.835,-179.903,7.854,149.463
C04356=1114.620,86.782,-56.817,-179.904,7.849,149.462
C04357=1114.625,86.534,-56.798,-179.906,7.845,149.462
C04358=1114.630,86.285,-56.780,-179.907,7.842,149.461
C04359=1114.636,86.035,-56.762,-179.908,7.838,149.461
C04360=1114.640,85.785,-56.743,-179.910,7.834,149.460
C04361=1114.645,85.537,-56.725,-179.910,7.831,149.460
C04362=1114.649,85.288,-56.707,-179.912,7.827,149.459
C04363=1114.654,85.038,-56.689,-179.913,7.823,149.459
C04364=1114.659,84.788,-56.670,-179.914,7.819,149.458
C04365=1114.664,84.539,-56.652,-179.915,7.815,149.458
C04366=1114.669,84.290,-56.634,-179.917,7.812,149.457
C04367=1114.674,84.041,-56.615,-179.917,7.808,149.456
C04368=1114.678,83.792,-56.597,-179.919,7.804,149.456
C04369=1114.683,83.542,-56.579,-179.920,7.800,149.455
C04370=1114.689,83.293,-56.560,-179.921,7.797,149.455
C04371=1114.694,83.044,-56.542,-179.922,7.793,149.454
C04372=1114.699,82.795,-56.524,-179.923,7.789,149.454
C04373=1114.703,82.545,-56.506,-179.924,7.785,149.453
C04374=1114.708,82.295,-56.488,-179.926,7.781,149.453
C04375=1114.713,82.046,-56.470,-179.926,7.778,149.452
C04376=1114.717,81.798,-56.451,-179.928,7.774,149.452
C04377=1114.722,81.549,-56.433,-179.929,7.770,149.451
C04378=1114.727,81.299,-56.415,-179.930,7.766,149.451
C04379=1114.731,81.049,-56.397,-179.931,7.763,149.450
C04380=1114.736,80.800,-56.379,-179.932,7.759,149.450
C04381=1114.742,80.551,-56.360,-179.933,7.755,149.449
C04382=1114.747,80.302,-56.342,-179.934,7.752,149.448
C04383=1114.752,80.052,-56.324,-179.935,7.747,149.448
C04384=1114.757,79.803,-56.306,-179.936,7.744,149.447
C04385=1114.761,79.553,-56.288,-179.937,7.740,149.447
C04386=1114.766,79.304,-56.270,-179.938,7.737,149.446
C04387=1114.771,79.055,-56.252,-179.940,7.733,149.446
C04388=1114.776,78.806,-56.234,-179.941,7.729,149.445
C04389=1114.781,78.556,-56.217,-179.942,7.725,149.445
C04390=1114.785,78.342,-56.201,-179.943,7.722,149.444
C04391=1114.789,78.128,-56.186,-179.944,7.719,149.444
C04392=1114.793,77.914,-56.170,-179.944,7.715,149.443
C04393=1114.797,77.700,-56.155,-179.944,7.713,149.443
C04394=1114.801,77.485,-56.140,-179.945,7.710,149.442
C04395=1114.805,77.271,-56.124,-179.946,7.707,149.442
C04396=1114.810,77.057,-56.109,-179.947,7.704,149.441
C04397=1114.814,76.843,-56.093,-179.948,7.700,149.441
C04398=1114.819,76.593,-56.075,-179.949,7.696,149.440
C04399=1114.824,76.344,-56.057,-179.951,7.693,149.440
C04400=1114.829,76.095,-56.039,-179.953,7.689,149.439
C04401=1114.834,75.846,-56.021,-179.954,7.684,149.439
C04402=1114.839,75.596,-56.004,-179.955,7.680,149.438
C04403=1114.843,75.347,-55.987,-179.957,7.677,149.438
C04404=1114.848,75.098,-55.969,-179.958,7.673,149.437
C04405=1114.853,74.849,-55.951,-179.960,7.668,149.437
C04406=1114.858,74.600,-55.933,-179.961,7.664,149.436
C04407=1114.863,74.350,-55.915,-179.963,7.661,149.436
C04408=1114.868,74.101,-55.897,-179.964,7.656,149.435
C04409=1114.872,73.851,-55.879,-179.965,7.652,149.435
C04410=1114.877,73.602,-55.861,-179.966,7.649,149.434
C04411=1114.882,73.352,-55.844,-179.968,7.645,149.434
C04412=1114.887,73.103,-55.827,-179.969,7.641,149.433
C04413=1114.892,72.854,-55.809,-179.971,7.637,149.433
C04414=1114.897,72.604,-55.791,-179.972,7.633,149.433
C04415=1114.902,72.355,-55.773,-179.974,7.629,149.432
C04416=1114.907,72.106,-55.755,-179.975,7.625,149.431
C04417=1114.911,71.857,-55.737,-179.976,7.621,149.431
C04418=1114.916,71.607,-55.721,-179.978,7.617,149.431
C04419=1114.921,71.358,-55.703,-179.979,7.613,149.430
C04420=1114.926,71.108,-55.685,-179.981,7.609,149.429
C04421=1114.931,70.859,-55.667,-179.982,7.605,149.429
C04422=1114.936,70.610,-55.649,-179.983,7.602,149.428
C04423=1114.940,70.360,-55.633,-179.984,7.598,149.428
C04424=1114.945,70.111,-55.615,-179.986,7.594,149.428
C04425=1114.951,69.862,-55.598,-179.987,7.590,149.427
C04426=1114.956,69.613,-55.580,-179.989,7.586,149.426
C04427=1114.961,69.363,-55.563,-179.990,7.582,149.426
C04428=1114.965,69.114,-55.545,-179.992,7.578,149.426
C04429=1114.970,68.865,-55.527,-179.993,7.574,149.425
C04430=1114.975,68.616,-55.511,-179.994,7.570,149.425
C04431=1114.980,68.366,-55.493,-179.996,7.566,149.424
C04432=1114.985,68.117,-55.475,-179.997,7.561,149.423
C04433=1114.990,67.867,-55.457,-179.998,7.558,149.423
C04434=1114.994,67.618,-55.441,-180.000,7.554,149.423
C04435=1115.000,67.368,-55.423,179.999,7.550,149.422
C04436=1115.004,67.119,-55.406,179.998,7.546,149.421
C04437=1115.009,66.869,-55.389,179.997,7.542,149.421
C04438=1115.014,66.620,-55.371,179.995,7.538,149.420
C04439=1115.020,66.371,-55.354,179.993,7.534,149.420
C04440=1115.024,66.122,-55.337,179.992,7.530,149.419
C04441=1115.029,65.872,-55.319,179.991,7.526,149.419
C04442=1115.034,65.623,-55.303,179.989,7.522,149.418
C04443=1115.038,65.374,-55.285,179.989,7.519,149.418
C04444=1115.044,65.124,-55.267,179.987,7.515,149.417
C04445=1115.048,64.875,-55.250,179.986,7.511,149.417
C04446=1115.053,64.661,-55.236,179.984,7.507,149.417
C04447=1115.056,64.446,-55.221,179.984,7.503,149.416
C04448=1115.061,64.232,-55.206,179.983,7.500,149.415
C04449=1115.066,64.018,-55.191,179.981,7.496,149.415
C04450=1115.069,63.804,-55.176,179.980,7.493,149.415
C04451=1115.074,63.590,-55.161,179.979,7.490,149.414
C04452=1115.078,63.375,-55.147,179.978,7.486,149.414
C04453=1115.082,63.161,-55.132,179.977,7.483,149.413
C04454=1115.087,62.911,-55.115,179.975,7.479,149.413
C04455=1115.092,62.662,-55.097,179.974,7.475,149.412
C04456=1115.097,62.413,-55.081,179.972,7.471,149.412
C04457=1115.102,62.163,-55.064,179.971,7.468,149.411
C04458=1115.106,61.914,-55.047,179.970,7.464,149.411
C04459=1115.111,61.665,-55.029,179.969,7.460,149.410
C04460=1115.116,61.415,-55.012,179.968,7.455,149.410
C04461=1115.122,61.166,-54.996,179.966,7.451,149.409
C04462=1115.126,60.917,-54.979,179.965,7.447,149.409
C04463=1115.131,60.667,-54.962,179.963,7.443,149.408
C04464=1115.136,60.418,-54.944,179.962,7.439,149.408
C04465=1115.141,60.168,-54.927,179.961,7.436,149.407
C04466=1115.146,59.919,-54.911,179.960,7.432,149.407
C04467=1115.151,59.670,-54.893,179.959,7.428,149.406
C04468=1115.156,59.420,-54.877,179.957,7.424,149.405
C04469=1115.161,59.170,-54.859,179.956,7.419,149.405
C04470=1115.166,58.922,-54.843,179.955,7.415,149.404
C04471=1115.170,58.672,-54.826,179.953,7.411,149.404
C04472=1115.176,58.422,-54.809,179.952,7.407,149.403
C04473=1115.180,58.173,-54.792,179.951,7.404,149.403
C04474=1115.186,57.924,-54.775,179.950,7.400,149.402
C04475=1115.190,57.675,-54.758,179.949,7.396,149.402
C04476=1115.194,57.425,-54.742,179.947,7.392,149.401
C04477=1115.200,57.176,-54.725,179.946,7.388,149.401
C04478=1115.205,56.927,-54.708,179.945,7.383,149.400
C04479=1115.210,56.677,-54.691,179.943,7.380,149.400
C04480=1115.214,56.427,-54.674,179.942,7.376,149.399
C04481=1115.220,56.179,-54.658,179.941,7.372,149.399
C04482=1115.225,55.929,-54.641,179.940,7.368,149.398
C04483=1115.229,55.679,-54.624,179.939,7.364,149.397
C04484=1115.234,55.431,-54.608,179.937,7.360,149.397
C04485=1115.240,55.181,-54.590,179.936,7.355,149.396
C04486=1115.244,54.931,-54.574,179.935,7.351,149.396
C04487=1115.249,54.682,-54.558,179.934,7.348,149.395
C04488=1115.255,54.432,-54.541,179.933,7.344,149.395
C04489=1115.259,54.183,-54.524,179.931,7.340,149.394
C04490=1115.264,53.934,-54.508,179.930,7.336,149.394
C04491=1115.269,53.684,-54.491,179.929,7.331,149.393
C04492=1115.274,53.435,-54.474,179.927,7.328,149.393
C04493=1115.279,53.186,-54.458,179.926,7.323,149.392
C04494=1115.283,52.936,-54.441,179.925,7.319,149.391
C04495=1115.290,52.687,-54.425,179.924,7.316,149.391
C04496=1115.294,52.437,-54.408,179.923,7.312,149.390
C04497=1115.299,52.188,-54.391,179.921,7.308,149.390
C04498=1115.304,51.939,-54.375,179.920,7.303,149.389
C04499=1115.309,51.689,-54.358,179.919,7.299,149.389
C04500=1115.314,51.440,-54.342,179.918,7.295,149.388
C04501=1115.319,51.190,-54.326,179.917,7.291,149.387
C04502=1115.323,50.977,-54.311,179.916,7.288,149.387
C04503=1115.328,50.762,-54.297,179.915,7.285,149.386
C04504=1115.331,50.547,-54.283,179.914,7.281,149.386
C04505=1115.335,50.333,-54.268,179.912,7.278,149.386
C04506=1115.340,50.119,-54.255,179.912,7.274,149.385
C04507=1115.344,49.904,-54.241,179.911,7.271,149.385
C04508=1115.349,49.690,-54.227,179.909,7.267,149.384
C04509=1115.352,49.475,-54.212,179.908,7.264,149.384
C04510=1115.358,49.226,-54.196,179.907,7.260,149.383
C04511=1115.362,48.977,-54.180,179.906,7.255,149.382
C04512=1115.367,48.728,-54.163,179.905,7.251,149.382
C04513=1115.372,48.478,-54.147,179.904,7.248,149.381
C04514=1115.377,48.229,-54.131,179.903,7.244,149.381
C04515=1115.382,47.979,-54.114,179.902,7.240,149.380
C04516=1115.388,47.730,-54.098,179.900,7.235,149.380
C04517=1115.392,47.480,-54.081,179.899,7.231,149.379
C04518=1115.397,47.231,-54.065,179.898,7.227,149.378
C04519=1115.402,46.981,-54.049,179.897,7.223,149.378
C04520=1115.407,46.732,-54.033,179.896,7.219,149.377
C04521=1115.412,46.482,-54.017,179.895,7.215,149.377
C04522=1115.417,46.233,-54.000,179.894,7.211,149.376
C04523=1115.422,45.984,-53.984,179.893,7.207,149.375
C04524=1115.426,45.734,-53.968,179.892,7.202,149.375
C04525=1115.431,45.485,-53.952,179.890,7.199,149.374
C04526=1115.436,45.235,-53.936,179.889,7.194,149.374
C04527=1115.441,44.986,-53.919,179.888,7.191,149.373
C04528=1115.446,44.736,-53.904,179.887,7.187,149.373
C04529=1115.451,44.487,-53.887,179.886,7.183,149.372
C04530=1115.456,44.237,-53.871,179.885,7.178,149.371
C04531=1115.461,43.989,-53.855,179.884,7.174,149.371
C04532=1115.466,43.739,-53.839,179.882,7.170,149.370
C04533=1115.471,43.490,-53.823,179.881,7.166,149.370
C04534=1115.476,43.240,-53.807,179.881,7.162,149.369
C04535=1115.481,42.990,-53.791,179.880,7.158,149.368
C04536=1115.486,42.741,-53.775,179.878,7.154,149.368
C04537=1115.491,42.491,-53.759,179.877,7.150,149.367
C04538=1115.496,42.243,-53.743,179.876,7.145,149.367
C04539=1115.501,41.992,-53.727,179.875,7.141,149.366
C04540=1115.506,41.744,-53.710,179.874,7.138,149.365
C04541=1115.511,41.494,-53.695,179.873,7.134,149.365
C04542=1115.516,41.244,-53.679,179.872,7.129,149.364
C04543=1115.521,40.995,-53.663,179.871,7.125,149.363
C04544=1115.526,40.745,-53.647,179.870,7.121,149.363
C04545=1115.531,40.496,-53.631,179.868,7.116,149.362
C04546=1115.536,40.247,-53.615,179.867,7.112,149.362
C04547=1115.541,39.997,-53.599,179.866,7.109,149.361
C04548=1115.546,39.748,-53.584,179.865,7.105,149.360
C04549=1115.550,39.498,-53.567,179.864,7.100,149.360
C04550=1115.556,39.249,-53.551,179.863,7.096,149.359
C04551=1115.561,39.000,-53.536,179.862,7.092,149.359
C04552=1115.566,38.749,-53.520,179.861,7.087,149.358
C04553=1115.571,38.501,-53.504,179.860,7.083,149.357
C04554=1115.576,38.251,-53.488,179.859,7.080,149.357
C04555=1115.581,38.001,-53.472,179.858,7.076,149.356
C04556=1115.586,37.752,-53.457,179.857,7.071,149.355
C04557=1115.591,37.503,-53.441,179.856,7.067,149.355
C04558=1115.596,37.288,-53.428,179.855,7.064,149.354
C04559=1115.600,37.074,-53.414,179.854,7.060,149.354
C04560=1115.604,36.860,-53.400,179.853,7.056,149.353
C04561=1115.608,36.645,-53.387,179.853,7.053,149.353
C04562=1115.613,36.431,-53.373,179.851,7.049,149.352
C04563=1115.617,36.216,-53.360,179.851,7.046,149.352
C04564=1115.622,36.002,-53.346,179.850,7.042,149.351
C04565=1115.626,35.787,-53.333,179.849,7.038,149.350
C04566=1115.630,35.538,-53.317,179.848,7.035,149.350
C04567=1115.635,35.288,-53.302,179.847,7.030,149.349
C04568=1115.641,35.039,-53.286,179.846,7.026,149.349
C04569=1115.645,34.789,-53.270,179.845,7.022,149.348
C04570=1115.650,34.540,-53.255,179.844,7.017,149.347
C04571=1115.655,34.291,-53.239,179.843,7.013,149.347
C04572=1115.661,34.042,-53.223,179.842,7.009,149.346
C04573=1115.665,33.791,-53.207,179.841,7.005,149.345
C04574=1115.670,33.542,-53.192,179.840,7.001,149.345
C04575=1115.675,33.293,-53.177,179.839,6.997,149.344
C04576=1115.680,33.043,-53.161,179.838,6.992,149.343
C04577=1115.685,32.794,-53.146,179.837,6.988,149.343
C04578=1115.690,32.544,-53.130,179.836,6.984,149.342
C04579=1115.696,32.295,-53.115,179.835,6.979,149.341
C04580=1115.700,32.046,-53.100,179.834,6.976,149.341
C04581=1115.705,31.796,-53.084,179.833,6.971,149.340
C04582=1115.710,31.546,-53.068,179.832,6.967,149.339
C04583=1115.715,31.297,-53.053,179.831,6.963,149.339
C04584=1115.720,31.048,-53.037,179.830,6.959,149.338
C04585=1115.725,30.798,-53.021,179.830,6.954,149.337
C04586=1115.730,30.549,-53.006,179.829,6.950,149.337
C04587=1115.735,30.299,-52.991,179.828,6.945,149.336
C04588=1115.740,30.050,-52.976,179.827,6.942,149.335
C04589=1115.746,29.800,-52.961,179.826,6.937,149.335
C04590=1115.750,29.550,-52.945,179.825,6.933,149.334
C04591=1115.755,29.301,-52.930,179.824,6.929,149.333
C04592=1115.760,29.051,-52.914,179.823,6.924,149.333
C04593=1115.765,28.802,-52.899,179.822,6.920,149.332
C04594=1115.773,28.427,-52.876,179.820,6.913,149.331
C04595=1115.780,28.052,-52.853,179.820,6.908,149.330
C04596=1115.788,27.677,-52.831,179.818,6.901,149.329
C04597=1115.795,27.302,-52.807,179.817,6.894,149.328
C04598=1115.801,27.052,-52.792,179.816,6.890,149.327
C04599=1115.805,26.803,-52.777,179.815,6.886,149.326
C04600=1115.811,26.553,-52.762,179.814,6.881,149.326
C04601=1115.816,26.304,-52.747,179.813,6.877,149.325
C04602=1115.821,26.055,-52.731,179.812,6.872,149.324
C04603=1115.825,25.805,-52.716,179.812,6.869,149.323
C04604=1115.831,25.555,-52.701,179.811,6.865,149.323
C04605=1115.835,25.306,-52.686,179.810,6.860,149.322
C04606=1115.841,25.056,-52.670,179.809,6.856,149.321
C04607=1115.846,24.807,-52.656,179.808,6.851,149.321
C04608=1115.851,24.557,-52.641,179.807,6.847,149.320
C04609=1115.856,24.308,-52.626,179.806,6.843,149.319
C04610=1115.860,24.059,-52.611,179.805,6.838,149.318
C04611=1115.866,23.809,-52.596,179.804,6.834,149.318
C04612=1115.871,23.560,-52.581,179.804,6.830,149.317
C04613=1115.876,23.310,-52.565,179.803,6.826,149.316
C04614=1115.882,23.006,-52.547,179.802,6.820,149.315
C04615=1115.888,22.703,-52.529,179.801,6.814,149.314
C04616=1115.894,22.399,-52.511,179.800,6.809,149.314
C04617=1115.899,22.096,-52.492,179.799,6.804,149.313
C04618=1115.905,21.846,-52.477,179.798,6.800,149.312
C04619=1115.910,21.597,-52.462,179.797,6.795,149.311
C04620=1115.916,21.347,-52.447,179.797,6.791,149.311
C04621=1115.920,21.098,-52.432,179.795,6.786,149.310
C04622=1115.925,20.848,-52.418,179.795,6.782,149.309
C04623=1115.931,20.599,-52.403,179.794,6.777,149.308
C04624=1115.935,20.349,-52.388,179.793,6.773,149.308
C04625=1115.940,20.100,-52.373,179.793,6.769,149.307
C04626=1115.945,19.851,-52.358,179.792,6.765,149.306
C04627=1115.950,19.601,-52.343,179.791,6.760,149.305
C04628=1115.955,19.352,-52.328,179.790,6.756,149.305
C04629=1115.961,19.102,-52.314,179.789,6.752,149.304
C04630=1115.966,18.852,-52.299,179.789,6.747,149.303
C04631=1115.970,18.603,-52.284,179.788,6.743,149.302
C04632=1115.976,18.353,-52.269,179.787,6.738,149.302
C04633=1115.981,18.104,-52.254,179.786,6.733,149.301
C04634=1115.986,17.854,-52.240,179.785,6.729,149.300
C04635=1115.990,17.605,-52.225,179.784,6.724,149.299
C04636=1115.996,17.355,-52.210,179.784,6.720,149.299
C04637=1116.001,17.106,-52.195,179.783,6.716,149.298
C04638=1116.006,16.856,-52.181,179.783,6.712,149.297
C04639=1116.011,16.607,-52.167,179.782,6.707,149.296
C04640=1116.016,16.357,-52.151,179.781,6.703,149.295
C04641=1116.021,16.107,-52.137,179.780,6.698,149.295
C04642=1116.026,15.858,-52.123,179.780,6.693,149.294
C04643=1116.031,15.609,-52.108,179.779,6.689,149.293
C04644=1116.037,15.359,-52.093,179.778,6.684,149.292
C04645=1116.042,15.110,-52.079,179.777,6.680,149.291
C04646=1116.046,14.861,-52.064,179.776,6.675,149.291
C04647=1116.051,14.611,-52.050,179.776,6.671,149.290
C04648=1116.056,14.361,-52.035,179.775,6.666,149.289
C04649=1116.062,14.112,-52.020,179.774,6.662,149.288
C04650=1116.067,13.862,-52.005,179.774,6.658,149.288
C04651=1116.072,13.612,-51.991,179.773,6.653,149.287
C04652=1116.077,13.363,-51.977,179.773,6.649,149.286
C04653=1116.081,13.113,-51.962,179.772,6.644,149.285
C04654=1116.086,12.864,-51.948,179.771,6.640,149.284
C04655=1116.092,12.615,-51.934,179.771,6.635,149.284
C04656=1116.097,12.365,-51.919,179.770,6.630,149.283
C04657=1116.102,12.116,-51.904,179.769,6.626,149.282
C04658=1116.107,11.866,-51.890,179.768,6.621,149.281
C04659=1116.112,11.616,-51.875,179.768,6.617,149.280
C04660=1116.117,11.367,-51.861,179.767,6.612,149.279
C04661=1116.122,11.117,-51.847,179.766,6.607,149.279
C04662=1116.127,10.868,-51.832,179.766,6.603,149.278
C04663=1116.132,10.619,-51.818,179.765,6.598,149.277
C04664=1116.137,10.369,-51.804,179.764,6.594,149.276
C04665=1116.142,10.119,-51.789,179.764,6.589,149.275
C04666=1116.147,9.904,-51.776,179.763,6.586,149.275
C04667=1116.151,9.690,-51.764,179.763,6.581,149.274
C04668=1116.155,9.475,-51.753,179.762,6.577,149.273
C04669=1116.160,9.260,-51.740,179.762,6.574,149.273
C04670=1116.164,9.046,-51.728,179.761,6.569,149.272
C04671=1116.168,8.832,-51.715,179.761,6.565,149.271
C04672=1116.173,8.617,-51.702,179.760,6.561,149.270
C04673=1116.178,8.402,-51.691,179.760,6.558,149.270
C04674=1116.183,8.152,-51.677,179.759,6.553,149.269
C04675=1116.187,7.903,-51.662,179.758,6.548,149.268
C04676=1116.192,7.653,-51.648,179.758,6.543,149.267
C04677=1116.198,7.405,-51.633,179.757,6.539,149.266
C04678=1116.203,7.155,-51.619,179.757,6.535,149.265
C04679=1116.208,6.905,-51.605,179.757,6.530,149.264
C04680=1116.213,6.655,-51.591,179.756,6.526,149.264
C04681=1116.218,6.406,-51.576,179.755,6.521,149.263
C04682=1116.223,6.157,-51.562,179.755,6.516,149.262
C04683=1116.228,5.907,-51.548,179.754,6.512,149.261
C04684=1116.233,5.657,-51.535,179.754,6.507,149.260
C04685=1116.238,5.407,-51.520,179.753,6.502,149.259
C04686=1116.244,5.158,-51.506,179.752,6.498,149.259
C04687=1116.249,4.908,-51.492,179.752,6.494,149.258
C04688=1116.253,4.659,-51.478,179.752,6.489,149.257
C04689=1116.258,4.409,-51.464,179.751,6.485,149.256
C04690=1116.263,4.160,-51.450,179.751,6.480,149.255
C04691=1116.268,3.910,-51.436,179.750,6.476,149.254
C04692=1116.273,3.661,-51.422,179.749,6.471,149.254
C04693=1116.278,3.411,-51.407,179.748,6.466,149.253
C04694=1116.284,3.162,-51.393,179.748,6.461,149.252
C04695=1116.289,2.912,-51.380,179.748,6.458,149.251
C04696=1116.294,2.662,-51.366,179.747,6.453,149.250
C04697=1116.299,2.413,-51.352,179.746,6.448,149.249
C04698=1116.304,2.164,-51.338,179.746,6.444,149.248
C04699=1116.309,1.914,-51.324,179.745,6.439,149.248
C04700=1116.314,1.665,-51.310,179.744,6.435,149.247
C04701=1116.320,1.415,-51.296,179.744,6.430,149.246
C04702=1116.325,1.165,-51.282,179.743,6.425,149.245
C04703=1116.330,0.915,-51.268,179.743,6.421,149.244
C04704=1116.334,0.666,-51.254,179.742,6.417,149.244
C04705=1116.339,0.417,-51.240,179.742,6.412,149.243
C04706=1116.345,0.166,-51.227,179.741,6.408,149.242
C04707=1116.350,-0.083,-51.213,179.740,6.403,149.241
C04708=1116.355,-0.332,-51.198,179.740,6.398,149.240
C04709=1116.360,-0.581,-51.185,179.739,6.394,149.239
C04710=1116.365,-0.831,-51.172,179.739,6.389,149.239
C04711=1116.370,-1.081,-51.157,179.738,6.385,149.238
C04712=1116.376,-1.330,-51.143,179.738,6.381,149.237
C04713=1116.380,-1.580,-51.130,179.737,6.376,149.236
C04714=1116.385,-1.830,-51.116,179.737,6.371,149.235
C04715=1116.391,-2.079,-51.102,179.736,6.367,149.235
C04716=1116.396,-2.329,-51.089,179.735,6.362,149.234
C04717=1116.400,-2.579,-51.075,179.735,6.358,149.233
C04718=1116.406,-2.828,-51.061,179.734,6.353,149.232
C04719=1116.411,-3.078,-51.047,179.733,6.349,149.231
C04720=1116.417,-3.327,-51.034,179.733,6.344,149.230
C04721=1116.421,-3.576,-51.020,179.732,6.340,149.230
C04722=1116.426,-3.791,-51.009,179.732,6.336,149.229
C04723=1116.430,-4.006,-50.997,179.731,6.332,149.228
C04724=1116.434,-4.220,-50.985,179.731,6.328,149.227
C04725=1116.438,-4.435,-50.973,179.730,6.324,149.227
C04726=1116.443,-4.650,-50.962,179.730,6.321,149.226
C04727=1116.447,-4.865,-50.949,179.729,6.316,149.225
C04728=1116.452,-5.079,-50.938,179.729,6.312,149.225
C04729=1116.456,-5.294,-50.926,179.728,6.309,149.224
C04730=1116.461,-5.543,-50.913,179.728,6.304,149.223
C04731=1116.467,-5.794,-50.899,179.727,6.300,149.222
C04732=1116.471,-6.043,-50.885,179.726,6.295,149.221
C04733=1116.477,-6.293,-50.872,179.726,6.290,149.221
C04734=1116.482,-6.542,-50.858,179.725,6.286,149.220
C04735=1116.487,-6.792,-50.845,179.724,6.281,149.219
C04736=1116.492,-7.041,-50.831,179.724,6.276,149.218
C04737=1116.497,-7.291,-50.818,179.723,6.272,149.217
C04738=1116.502,-7.540,-50.804,179.723,6.268,149.217
C04739=1116.508,-7.790,-50.791,179.722,6.263,149.216
C04740=1116.512,-8.040,-50.777,179.722,6.259,149.215
C04741=1116.518,-8.289,-50.764,179.721,6.254,149.214
C04742=1116.522,-8.539,-50.751,179.720,6.250,149.213
C04743=1116.528,-8.788,-50.737,179.720,6.245,149.212
C04744=1116.533,-9.038,-50.724,179.719,6.241,149.212
C04745=1116.538,-9.287,-50.710,179.718,6.236,149.211
C04746=1116.543,-9.538,-50.697,179.718,6.231,149.210
C04747=1116.548,-9.787,-50.684,179.717,6.226,149.209
C04748=1116.553,-10.037,-50.670,179.716,6.222,149.208
C04749=1116.559,-10.286,-50.657,179.716,6.217,149.207
C04750=1116.563,-10.536,-50.643,179.715,6.213,149.207
C04751=1116.569,-10.785,-50.630,179.715,6.209,149.206
C04752=1116.574,-11.035,-50.617,179.714,6.204,149.205
C04753=1116.579,-11.284,-50.603,179.714,6.200,149.204
C04754=1116.584,-11.534,-50.590,179.713,6.195,149.203
C04755=1116.589,-11.784,-50.577,179.712,6.191,149.203
C04756=1116.595,-12.033,-50.563,179.712,6.186,149.202
C04757=1116.599,-12.283,-50.550,179.711,6.181,149.201
C04758=1116.605,-12.532,-50.537,179.710,6.177,149.200
C04759=1116.610,-12.782,-50.524,179.710,6.172,149.199
C04760=1116.615,-13.031,-50.510,179.709,6.167,149.198
C04761=1116.620,-13.281,-50.497,179.709,6.163,149.197
C04762=1116.625,-13.531,-50.485,179.708,6.158,149.197
C04763=1116.630,-13.781,-50.471,179.708,6.154,149.196
C04764=1116.635,-14.030,-50.458,179.707,6.149,149.195
C04765=1116.641,-14.279,-50.445,179.707,6.144,149.194
C04766=1116.645,-14.529,-50.432,179.706,6.140,149.193
C04767=1116.651,-14.779,-50.419,179.705,6.135,149.192
C04768=1116.656,-15.029,-50.406,179.705,6.130,149.192
C04769=1116.660,-15.278,-50.392,179.704,6.126,149.191
C04770=1116.666,-15.527,-50.379,179.703,6.121,149.190
C04771=1116.671,-15.777,-50.366,179.703,6.117,149.189
C04772=1116.676,-16.027,-50.353,179.702,6.112,149.188
C04773=1116.682,-16.276,-50.340,179.702,6.107,149.187
C04774=1116.686,-16.526,-50.327,179.701,6.102,149.186
C04775=1116.692,-16.776,-50.314,179.700,6.098,149.186
C04776=1116.697,-17.025,-50.302,179.700,6.093,149.185
C04777=1116.701,-17.275,-50.288,179.699,6.089,149.184
C04778=1116.707,-17.490,-50.277,179.699,6.085,149.183
C04779=1116.711,-17.704,-50.266,179.698,6.080,149.182
C04780=1116.715,-17.919,-50.255,179.698,6.077,149.182
C04781=1116.720,-18.134,-50.244,179.697,6.072,149.181
C04782=1116.724,-18.348,-50.232,179.697,6.069,149.180
C04783=1116.728,-18.564,-50.221,179.696,6.064,149.180
C04784=1116.733,-18.778,-50.211,179.696,6.061,149.179
C04785=1116.738,-18.993,-50.199,179.695,6.057,149.178
C04786=1116.742,-19.243,-50.186,179.694,6.051,149.177
C04787=1116.748,-19.493,-50.173,179.694,6.047,149.176
C04788=1116.753,-19.742,-50.160,179.693,6.042,149.175
C04789=1116.758,-19.992,-50.147,179.693,6.037,149.175
C04790=1116.763,-20.241,-50.135,179.692,6.033,149.174
C04791=1116.769,-20.491,-50.122,179.691,6.028,149.173
C04792=1116.774,-20.740,-50.109,179.691,6.023,149.172
C04793=1116.778,-20.990,-50.096,179.690,6.019,149.171
C04794=1116.783,-21.240,-50.083,179.690,6.014,149.170
C04795=1116.789,-21.489,-50.070,179.689,6.009,149.169
C04796=1116.794,-21.739,-50.058,179.689,6.005,149.169
C04797=1116.799,-21.989,-50.045,179.688,6.000,149.168
C04798=1116.804,-22.238,-50.032,179.688,5.995,149.167
C04799=1116.809,-22.487,-50.020,179.687,5.990,149.166
C04800=1116.815,-22.737,-50.007,179.687,5.986,149.165
C04801=1116.820,-22.987,-49.994,179.686,5.980,149.164
C04802=1116.825,-23.237,-49.981,179.685,5.976,149.163
C04803=1116.830,-23.486,-49.969,179.684,5.971,149.163
C04804=1116.835,-23.735,-49.956,179.684,5.966,149.162
C04805=1116.840,-23.986,-49.943,179.684,5.962,149.161
C04806=1116.846,-24.235,-49.930,179.683,5.957,149.160
C04807=1116.851,-24.485,-49.918,179.683,5.952,149.159
C04808=1116.856,-24.734,-49.906,179.682,5.947,149.158
C04809=1116.861,-24.984,-49.893,179.682,5.943,149.157
C04810=1116.866,-25.234,-49.880,179.681,5.937,149.156
C04811=1116.871,-25.483,-49.867,179.680,5.932,149.155
C04812=1116.876,-25.733,-49.856,179.680,5.928,149.154
C04813=1116.882,-25.983,-49.842,179.680,5.923,149.153
C04814=1116.887,-26.232,-49.830,179.681,5.919,149.152
C04815=1116.892,-26.482,-49.817,179.681,5.915,149.151
C04816=1116.897,-26.732,-49.805,179.682,5.911,149.150
C04817=1116.902,-26.981,-49.792,179.682,5.906,149.149
C04818=1116.908,-27.230,-49.780,179.682,5.902,149.148
C04819=1116.913,-27.480,-49.768,179.683,5.898,149.147
C04820=1116.918,-27.730,-49.755,179.683,5.893,149.146
C04821=1116.923,-27.980,-49.742,179.683,5.889,149.145
C04822=1116.928,-28.229,-49.730,179.683,5.885,149.144
C04823=1116.933,-28.479,-49.718,179.684,5.881,149.143
C04824=1116.938,-28.728,-49.705,179.684,5.877,149.142
C04825=1116.943,-28.978,-49.693,179.685,5.873,149.141
C04826=1116.949,-29.228,-49.681,179.684,5.868,149.140
C04827=1116.953,-29.478,-49.668,179.684,5.864,149.139
C04828=1116.958,-29.727,-49.655,179.684,5.860,149.138
C04829=1116.964,-29.977,-49.643,179.684,5.855,149.137
C04830=1116.969,-30.226,-49.631,179.685,5.851,149.136
C04831=1116.975,-30.476,-49.617,179.685,5.847,149.135
C04832=1116.980,-30.726,-49.606,179.684,5.842,149.134
C04833=1116.985,-30.975,-49.593,179.684,5.838,149.133
C04834=1116.989,-31.191,-49.583,179.685,5.834,149.132
C04835=1116.993,-31.405,-49.572,179.684,5.831,149.132
C04836=1116.998,-31.620,-49.561,179.684,5.827,149.131
C04837=1117.002,-31.834,-49.551,179.684,5.823,149.130
C04838=1117.007,-32.049,-49.540,179.684,5.819,149.129
C04839=1117.012,-32.264,-49.530,179.684,5.816,149.129
C04840=1117.016,-32.480,-49.518,179.683,5.812,149.128
C04841=1117.020,-32.694,-49.508,179.684,5.808,149.127
C04842=1117.025,-32.944,-49.496,179.683,5.804,149.126
C04843=1117.031,-33.194,-49.484,179.683,5.799,149.125
C04844=1117.036,-33.443,-49.471,179.682,5.795,149.125
C04845=1117.041,-33.693,-49.459,179.682,5.790,149.124
C04846=1117.046,-33.942,-49.447,179.681,5.786,149.123
C04847=1117.052,-34.192,-49.435,179.681,5.781,149.122
C04848=1117.057,-34.442,-49.422,179.681,5.776,149.121
C04849=1117.062,-34.691,-49.410,179.681,5.772,149.120
C04850=1117.068,-34.941,-49.398,179.680,5.768,149.119
C04851=1117.072,-35.191,-49.385,179.679,5.763,149.118
C04852=1117.077,-35.440,-49.373,179.679,5.758,149.118
C04853=1117.082,-35.690,-49.362,179.678,5.754,149.117
C04854=1117.087,-35.940,-49.349,179.677,5.749,149.116
C04855=1117.093,-36.190,-49.337,179.677,5.745,149.115
C04856=1117.098,-36.439,-49.324,179.677,5.740,149.114
C04857=1117.103,-36.689,-49.313,179.676,5.736,149.113
C04858=1117.109,-36.939,-49.301,179.675,5.730,149.113
C04859=1117.114,-37.188,-49.288,179.674,5.725,149.112
C04860=1117.119,-37.438,-49.277,179.673,5.721,149.111
C04861=1117.124,-37.687,-49.264,179.673,5.716,149.110
C04862=1117.129,-37.937,-49.252,179.672,5.711,149.109
C04863=1117.135,-38.187,-49.240,179.671,5.706,149.109
C04864=1117.140,-38.436,-49.228,179.670,5.702,149.108
C04865=1117.145,-38.686,-49.216,179.669,5.696,149.107
C04866=1117.150,-38.936,-49.205,179.668,5.692,149.106
C04867=1117.155,-39.185,-49.192,179.667,5.686,149.105
C04868=1117.160,-39.435,-49.180,179.666,5.682,149.104
C04869=1117.166,-39.685,-49.168,179.665,5.676,149.104
C04870=1117.171,-39.934,-49.156,179.665,5.671,149.103
C04871=1117.176,-40.184,-49.144,179.663,5.666,149.102
C04872=1117.181,-40.434,-49.133,179.662,5.661,149.101
C04873=1117.187,-40.683,-49.121,179.662,5.656,149.100
C04874=1117.192,-40.932,-49.108,179.660,5.651,149.099
C04875=1117.197,-41.182,-49.097,179.659,5.645,149.099
C04876=1117.202,-41.432,-49.085,179.658,5.640,149.098
C04877=1117.208,-41.682,-49.073,179.657,5.635,149.097
C04878=1117.212,-41.932,-49.062,179.656,5.630,149.096
C04879=1117.218,-42.181,-49.049,179.655,5.624,149.095
C04880=1117.223,-42.431,-49.038,179.654,5.619,149.095
C04881=1117.228,-42.680,-49.026,179.653,5.614,149.094
C04882=1117.233,-42.930,-49.014,179.652,5.608,149.093
C04883=1117.239,-43.180,-49.003,179.651,5.603,149.092
C04884=1117.244,-43.429,-48.992,179.651,5.598,149.091
C04885=1117.249,-43.679,-48.980,179.652,5.594,149.090
C04886=1117.255,-43.929,-48.968,179.652,5.589,149.088
C04887=1117.259,-44.178,-48.956,179.652,5.584,149.087
C04888=1117.264,-44.428,-48.944,179.652,5.580,149.086
C04889=1117.270,-44.678,-48.932,179.652,5.574,149.085
C04890=1117.274,-44.893,-48.922,179.653,5.571,149.084
C04891=1117.279,-45.108,-48.912,179.653,5.567,149.083
C04892=1117.283,-45.323,-48.903,179.653,5.563,149.082
C04893=1117.288,-45.538,-48.893,179.653,5.559,149.082
C04894=1117.292,-45.753,-48.883,179.653,5.555,149.081
C04895=1117.297,-45.968,-48.872,179.653,5.551,149.080
C04896=1117.301,-46.183,-48.862,179.653,5.546,149.079
C04897=1117.306,-46.398,-48.852,179.653,5.542,149.078
C04898=1117.310,-46.647,-48.841,179.654,5.538,149.077
C04899=1117.316,-46.897,-48.829,179.654,5.533,149.076
C04900=1117.322,-47.147,-48.817,179.653,5.528,149.075
C04901=1117.327,-47.396,-48.806,179.654,5.524,149.074
C04902=1117.332,-47.646,-48.794,179.654,5.518,149.072
C04903=1117.337,-47.896,-48.783,179.655,5.514,149.071
C04904=1117.343,-48.145,-48.771,179.654,5.509,149.070
C04905=1117.347,-48.395,-48.760,179.654,5.504,149.069
C04906=1117.353,-48.645,-48.748,179.655,5.500,149.068
C04907=1117.357,-48.894,-48.737,179.655,5.495,149.067
C04908=1117.363,-49.144,-48.725,179.655,5.491,149.066
C04909=1117.368,-49.393,-48.714,179.655,5.486,149.065
C04910=1117.374,-49.643,-48.702,179.656,5.481,149.064
C04911=1117.378,-49.893,-48.691,179.656,5.477,149.063
C04912=1117.384,-50.143,-48.680,179.656,5.471,149.062
C04913=1117.389,-50.393,-48.668,179.656,5.467,149.060
C04914=1117.395,-50.642,-48.657,179.656,5.462,149.060
C04915=1117.400,-50.892,-48.645,179.656,5.457,149.058
C04916=1117.405,-51.142,-48.634,179.657,5.453,149.057
C04917=1117.410,-51.391,-48.623,179.656,5.448,149.056
C04918=1117.416,-51.641,-48.611,179.657,5.444,149.055
C04919=1117.420,-51.890,-48.600,179.657,5.439,149.054
C04920=1117.426,-52.140,-48.588,179.657,5.434,149.053
C04921=1117.431,-52.390,-48.577,179.657,5.430,149.052
C04922=1117.437,-52.640,-48.566,179.658,5.424,149.051
C04923=1117.441,-52.889,-48.554,179.658,5.420,149.050
C04924=1117.447,-53.139,-48.543,179.658,5.415,149.049
C04925=1117.452,-53.389,-48.531,179.658,5.410,149.048
C04926=1117.458,-53.638,-48.520,179.659,5.406,149.046
C04927=1117.463,-53.888,-48.509,179.658,5.401,149.046
C04928=1117.467,-54.138,-48.498,179.659,5.397,149.044
C04929=1117.473,-54.388,-48.486,179.659,5.392,149.043
C04930=1117.478,-54.637,-48.475,179.659,5.387,149.042
C04931=1117.484,-54.887,-48.464,179.659,5.383,149.041
C04932=1117.488,-55.137,-48.453,179.659,5.377,149.040
C04933=1117.494,-55.386,-48.442,179.659,5.373,149.039
C04934=1117.499,-55.636,-48.430,179.660,5.368,149.038
C04935=1117.504,-55.885,-48.419,179.659,5.364,149.037
C04936=1117.510,-56.136,-48.407,179.660,5.359,149.036
C04937=1117.515,-56.385,-48.396,179.660,5.354,149.035
C04938=1117.520,-56.635,-48.385,179.660,5.350,149.034
C04939=1117.525,-56.885,-48.374,179.660,5.345,149.033
C04940=1117.531,-57.134,-48.363,179.660,5.340,149.031
C04941=1117.535,-57.384,-48.352,179.661,5.336,149.031
C04942=1117.541,-57.634,-48.340,179.661,5.331,149.029
C04943=1117.546,-57.883,-48.330,179.661,5.326,149.028
C04944=1117.551,-58.133,-48.318,179.661,5.322,149.027
C04945=1117.556,-58.383,-48.307,179.662,5.317,149.026
C04946=1117.561,-58.598,-48.297,179.661,5.313,149.025
C04947=1117.565,-58.813,-48.288,179.661,5.309,149.024
C04948=1117.570,-59.027,-48.279,179.662,5.305,149.023
C04949=1117.574,-59.242,-48.269,179.662,5.301,149.022
C04950=1117.579,-59.458,-48.260,179.662,5.297,149.022
C04951=1117.583,-59.673,-48.250,179.662,5.293,149.021
C04952=1117.588,-59.888,-48.240,179.662,5.289,149.020
C04953=1117.592,-60.103,-48.230,179.663,5.285,149.019
C04954=1117.598,-60.353,-48.220,179.662,5.279,149.018
C04955=1117.603,-60.602,-48.209,179.661,5.275,149.017
C04956=1117.608,-60.853,-48.198,179.660,5.269,149.016
C04957=1117.614,-61.102,-48.187,179.660,5.264,149.015
C04958=1117.618,-61.351,-48.175,179.659,5.259,149.014
C04959=1117.624,-61.601,-48.165,179.658,5.254,149.013
C04960=1117.629,-61.851,-48.153,179.658,5.249,149.012
C04961=1117.634,-62.101,-48.143,179.657,5.244,149.011
C04962=1117.640,-62.350,-48.132,179.657,5.239,149.011
C04963=1117.645,-62.600,-48.121,179.656,5.233,149.009
C04964=1117.650,-62.849,-48.110,179.656,5.228,149.008
C04965=1117.656,-63.100,-48.099,179.655,5.223,149.008
C04966=1117.660,-63.349,-48.088,179.654,5.218,149.007
C04967=1117.666,-63.599,-48.078,179.654,5.213,149.006
C04968=1117.671,-63.848,-48.066,179.654,5.207,149.005
C04969=1117.676,-64.098,-48.056,179.653,5.202,149.004
C04970=1117.682,-64.348,-48.044,179.652,5.197,149.003
C04971=1117.687,-64.598,-48.034,179.652,5.192,149.002
C04972=1117.692,-64.848,-48.023,179.652,5.187,149.001
C04973=1117.698,-65.097,-48.013,179.651,5.181,149.000
C04974=1117.703,-65.347,-48.002,179.651,5.176,148.999
C04975=1117.707,-65.597,-47.991,179.650,5.171,148.998
C04976=1117.713,-65.846,-47.980,179.650,5.166,148.997
C04977=1117.719,-66.097,-47.969,179.650,5.161,148.996
C04978=1117.724,-66.346,-47.958,179.649,5.155,148.995
C04979=1117.729,-66.596,-47.948,179.649,5.150,148.993
C04980=1117.734,-66.845,-47.938,179.649,5.145,148.993
C04981=1117.739,-67.095,-47.926,179.648,5.140,148.992
C04982=1117.745,-67.345,-47.916,179.648,5.135,148.990
C04983=1117.750,-67.595,-47.906,179.647,5.130,148.990
C04984=1117.755,-67.844,-47.895,179.647,5.124,148.988
C04985=1117.760,-68.094,-47.884,179.647,5.119,148.987
C04986=1117.766,-68.343,-47.874,179.647,5.114,148.986
C04987=1117.771,-68.592,-47.863,179.646,5.108,148.985
C04988=1117.776,-68.843,-47.852,179.646,5.103,148.984
C04989=1117.781,-69.092,-47.842,179.646,5.098,148.983
C04990=1117.786,-69.342,-47.832,179.645,5.093,148.982
C04991=1117.792,-69.591,-47.821,179.645,5.087,148.981
C04992=1117.797,-69.842,-47.810,179.645,5.083,148.980
C04993=1117.803,-70.091,-47.799,179.645,5.077,148.979
C04994=1117.808,-70.342,-47.789,179.645,5.072,148.978
C04995=1117.814,-70.591,-47.778,179.644,5.067,148.977
C04996=1117.819,-70.840,-47.768,179.644,5.062,148.976
C04997=1117.823,-71.090,-47.758,179.644,5.056,148.974
C04998=1117.829,-71.340,-47.747,179.643,5.051,148.974
C04999=1117.834,-71.590,-47.737,179.644,5.046,148.972
C05000=1117.839,-71.839,-47.727,179.644,5.041,148.971
C05001=1117.845,-72.089,-47.716,179.644,5.035,148.970
C05002=1117.850,-72.304,-47.707,179.644,5.031,148.969
C05003=1117.854,-72.520,-47.698,179.643,5.026,148.968
C05004=1117.858,-72.735,-47.689,179.643,5.022,148.967
C05005=1117.863,-72.950,-47.680,179.643,5.017,148.966
C05006=1117.867,-73.165,-47.671,179.643,5.012,148.965
C05007=1117.872,-73.381,-47.662,179.643,5.008,148.964
C05008=1117.877,-73.595,-47.653,179.643,5.004,148.964
C05009=1117.881,-73.811,-47.645,179.643,5.000,148.963
C05010=1117.887,-74.060,-47.634,179.642,4.994,148.961
C05011=1117.891,-74.310,-47.623,179.642,4.989,148.960
C05012=1117.897,-74.559,-47.613,179.643,4.984,148.959
C05013=1117.903,-74.809,-47.603,179.643,4.978,148.958
C05014=1117.908,-75.059,-47.592,179.643,4.973,148.957
C05015=1117.913,-75.309,-47.582,179.643,4.968,148.956
C05016=1117.919,-75.558,-47.572,179.643,4.963,148.955
C05017=1117.923,-75.808,-47.562,179.642,4.957,148.954
C05018=1117.929,-76.058,-47.551,179.642,4.952,148.952
C05019=1117.934,-76.307,-47.541,179.643,4.947,148.951
C05020=1117.939,-76.557,-47.531,179.643,4.942,148.950
C05021=1117.945,-76.807,-47.520,179.643,4.937,148.949
C05022=1117.951,-77.057,-47.511,179.643,4.932,148.948
C05023=1117.956,-77.306,-47.501,179.643,4.926,148.947
C05024=1117.961,-77.557,-47.491,179.643,4.921,148.945
C05025=1117.966,-77.806,-47.481,179.643,4.916,148.944
C05026=1117.972,-78.056,-47.470,179.644,4.911,148.943
C05027=1117.977,-78.306,-47.460,179.644,4.906,148.942
C05028=1117.982,-78.555,-47.450,179.644,4.901,148.941
C05029=1117.987,-78.805,-47.440,179.644,4.896,148.940
C05030=1117.993,-79.054,-47.430,179.644,4.890,148.938
C05031=1117.998,-79.304,-47.419,179.644,4.885,148.937
C05032=1118.004,-79.554,-47.409,179.645,4.880,148.936
C05033=1118.009,-79.804,-47.400,179.645,4.875,148.935
C05034=1118.014,-80.053,-47.390,179.645,4.870,148.934
C05035=1118.019,-80.304,-47.379,179.645,4.865,148.933
C05036=1118.025,-80.553,-47.369,179.645,4.859,148.931
C05037=1118.030,-80.802,-47.359,179.645,4.854,148.930
C05038=1118.035,-81.053,-47.349,179.646,4.849,148.929
C05039=1118.041,-81.303,-47.339,179.646,4.844,148.928
C05040=1118.046,-81.552,-47.329,179.646,4.839,148.927
C05041=1118.051,-81.802,-47.320,179.646,4.834,148.925
C05042=1118.057,-82.051,-47.309,179.646,4.829,148.924
C05043=1118.062,-82.301,-47.299,179.646,4.823,148.923
C05044=1118.067,-82.551,-47.290,179.647,4.818,148.922
C05045=1118.072,-82.801,-47.280,179.647,4.813,148.921
C05046=1118.078,-83.050,-47.269,179.647,4.808,148.920
C05047=1118.083,-83.301,-47.259,179.648,4.804,148.918
C05048=1118.088,-83.550,-47.250,179.648,4.798,148.917
C05049=1118.094,-83.800,-47.240,179.649,4.793,148.916
C05050=1118.099,-84.050,-47.230,179.649,4.788,148.915
C05051=1118.104,-84.299,-47.220,179.649,4.783,148.913
C05052=1118.110,-84.550,-47.210,179.649,4.777,148.912
C05053=1118.114,-84.799,-47.201,179.650,4.773,148.911
C05054=1118.120,-85.048,-47.190,179.650,4.768,148.910
C05055=1118.126,-85.299,-47.181,179.650,4.763,148.909
C05056=1118.131,-85.548,-47.171,179.651,4.757,148.907
C05057=1118.136,-85.798,-47.161,179.651,4.752,148.906
C05058=1118.141,-86.013,-47.153,179.651,4.748,148.905
C05059=1118.145,-86.229,-47.144,179.652,4.744,148.904
C05060=1118.150,-86.443,-47.135,179.652,4.740,148.903
C05061=1118.154,-86.659,-47.127,179.653,4.736,148.902
C05062=1118.159,-86.874,-47.118,179.653,4.731,148.901
C05063=1118.163,-87.089,-47.111,179.653,4.727,148.900
C05064=1118.168,-87.304,-47.102,179.654,4.722,148.899
C05065=1118.173,-87.520,-47.094,179.654,4.718,148.898
C05066=1118.178,-87.769,-47.084,179.654,4.713,148.897
C05067=1118.183,-88.019,-47.074,179.655,4.708,148.895
C05068=1118.189,-88.269,-47.065,179.656,4.703,148.894
C05069=1118.194,-88.518,-47.055,179.656,4.698,148.893
C05070=1118.200,-88.768,-47.045,179.656,4.693,148.892
C05071=1118.204,-89.018,-47.035,179.657,4.689,148.891
C05072=1118.210,-89.268,-47.025,179.657,4.683,148.889
C05073=1118.215,-89.518,-47.016,179.658,4.678,148.888
C05074=1118.221,-89.767,-47.006,179.659,4.674,148.887
C05075=1118.226,-90.017,-46.997,179.659,4.668,148.886
C05076=1118.231,-90.267,-46.987,179.659,4.664,148.884
C05077=1118.237,-90.517,-46.978,179.660,4.659,148.883
C05078=1118.242,-90.766,-46.968,179.661,4.654,148.882
C05079=1118.247,-91.017,-46.958,179.661,4.649,148.881
C05080=1118.252,-91.266,-46.948,179.661,4.644,148.879
C05081=1118.258,-91.516,-46.939,179.662,4.640,148.878
C05082=1118.263,-91.766,-46.929,179.662,4.634,148.877
C05083=1118.268,-92.015,-46.920,179.664,4.630,148.876
C05084=1118.274,-92.265,-46.910,179.664,4.624,148.874
C05085=1118.279,-92.515,-46.901,179.665,4.620,148.873
C05086=1118.285,-92.764,-46.891,179.665,4.615,148.872
C05087=1118.290,-93.014,-46.882,179.666,4.611,148.871
C05088=1118.295,-93.264,-46.872,179.666,4.606,148.870
C05089=1118.301,-93.514,-46.863,179.667,4.601,148.868
C05090=1118.306,-93.763,-46.853,179.668,4.596,148.867
C05091=1118.311,-94.014,-46.843,179.668,4.591,148.866
C05092=1118.316,-94.263,-46.833,179.669,4.587,148.865
C05093=1118.322,-94.513,-46.824,179.669,4.582,148.864
C05094=1118.326,-94.762,-46.815,179.670,4.577,148.862
C05095=1118.332,-95.012,-46.805,179.670,4.572,148.861
C05096=1118.337,-95.262,-46.796,179.670,4.567,148.860
C05097=1118.343,-95.512,-46.786,179.670,4.562,148.859
C05098=1118.348,-95.762,-46.777,179.671,4.558,148.858
C05099=1118.354,-96.011,-46.767,179.671,4.552,148.856
C05100=1118.359,-96.261,-46.758,179.672,4.547,148.855
C05101=1118.364,-96.511,-46.749,179.672,4.542,148.854
C05102=1118.370,-96.761,-46.739,179.673,4.538,148.853
C05103=1118.375,-97.010,-46.730,179.673,4.533,148.852
C05104=1118.381,-97.261,-46.721,179.673,4.527,148.851
C05105=1118.386,-97.510,-46.711,179.673,4.522,148.849
C05106=1118.391,-97.760,-46.702,179.674,4.518,148.848
C05107=1118.397,-98.010,-46.693,179.674,4.513,148.847
C05108=1118.402,-98.259,-46.683,179.674,4.508,148.846
C05109=1118.408,-98.509,-46.673,179.674,4.503,148.845
C05110=1118.413,-98.759,-46.665,179.675,4.498,148.844
C05111=1118.418,-99.008,-46.655,179.675,4.493,148.842
C05112=1118.423,-99.258,-46.645,179.676,4.488,148.841
C05113=1118.429,-99.508,-46.637,179.676,4.483,148.840
C05114=1118.433,-99.723,-46.629,179.676,4.479,148.839
C05115=1118.437,-99.939,-46.620,179.677,4.475,148.838
C05116=1118.442,-100.154,-46.613,179.677,4.470,148.837
C05117=1118.447,-100.370,-46.604,179.677,4.466,148.836
C05118=1118.452,-100.585,-46.596,179.677,4.462,148.835
C05119=1118.457,-100.800,-46.589,179.677,4.457,148.834
C05120=1118.461,-101.015,-46.580,179.678,4.453,148.833
C05121=1118.465,-101.230,-46.573,179.678,4.449,148.832
C05122=1118.471,-101.480,-46.564,179.678,4.444,148.831
C05123=1118.477,-101.730,-46.554,179.678,4.438,148.830
C05124=1118.482,-101.980,-46.545,179.679,4.433,148.828
C05125=1118.487,-102.229,-46.536,179.679,4.429,148.827
C05126=1118.492,-102.479,-46.527,179.680,4.424,148.826
C05127=1118.498,-102.729,-46.517,179.680,4.419,148.825
C05128=1118.503,-102.979,-46.508,179.680,4.413,148.824
C05129=1118.508,-103.229,-46.499,179.680,4.408,148.822
C05130=1118.513,-103.478,-46.490,179.681,4.403,148.821
C05131=1118.519,-103.728,-46.480,179.681,4.398,148.820
C05132=1118.524,-103.978,-46.471,179.682,4.394,148.819
C05133=1118.530,-104.227,-46.463,179.682,4.388,148.818
C05134=1118.535,-104.477,-46.454,179.682,4.384,148.817
C05135=1118.541,-104.727,-46.445,179.682,4.378,148.815
C05136=1118.546,-104.977,-46.436,179.682,4.373,148.814
C05137=1118.551,-105.227,-46.427,179.682,4.368,148.813
C05138=1118.556,-105.476,-46.417,179.683,4.363,148.812
C05139=1118.561,-105.726,-46.408,179.683,4.359,148.811
C05140=1118.567,-105.976,-46.399,179.684,4.353,148.809
C05141=1118.572,-106.226,-46.390,179.684,4.348,148.808
C05142=1118.577,-106.476,-46.381,179.684,4.343,148.807
C05143=1118.583,-106.725,-46.372,179.684,4.338,148.806
C05144=1118.588,-106.975,-46.363,179.685,4.333,148.805
C05145=1118.594,-107.225,-46.354,179.685,4.328,148.804
C05146=1118.599,-107.475,-46.345,179.685,4.322,148.802
C05147=1118.604,-107.725,-46.336,179.685,4.317,148.801
C05148=1118.610,-107.975,-46.327,179.686,4.312,148.800
C05149=1118.615,-108.225,-46.318,179.686,4.307,148.799
C05150=1118.621,-108.474,-46.310,179.687,4.303,148.798
C05151=1118.626,-108.724,-46.301,179.687,4.297,148.796
C05152=1118.632,-108.974,-46.291,179.687,4.292,148.795
C05153=1118.637,-109.224,-46.283,179.687,4.287,148.794
C05154=1118.642,-109.474,-46.274,179.688,4.282,148.793
C05155=1118.647,-109.723,-46.265,179.688,4.277,148.792
C05156=1118.653,-109.973,-46.256,179.688,4.272,148.790
C05157=1118.658,-110.222,-46.247,179.688,4.266,148.789
C05158=1118.663,-110.472,-46.238,179.689,4.261,148.788
C05159=1118.668,-110.722,-46.230,179.689,4.256,148.787
C05160=1118.674,-110.972,-46.221,179.689,4.251,148.786
C05161=1118.679,-111.221,-46.212,179.689,4.246,148.784
C05162=1118.685,-111.471,-46.203,179.690,4.241,148.783
C05163=1118.691,-111.722,-46.194,179.690,4.235,148.782
C05164=1118.696,-111.972,-46.186,179.690,4.230,148.781
C05165=1118.701,-112.221,-46.177,179.690,4.225,148.780
C05166=1118.707,-112.471,-46.168,179.691,4.220,148.778
C05167=1118.712,-112.720,-46.159,179.691,4.215,148.777
C05168=1118.717,-112.970,-46.150,179.691,4.210,148.776
C05169=1118.722,-113.220,-46.141,179.691,4.204,148.775
C05170=1118.727,-113.435,-46.134,179.692,4.200,148.773
C05171=1118.732,-113.651,-46.127,179.692,4.195,148.773
C05172=1118.737,-113.866,-46.119,179.692,4.191,148.772
C05173=1118.741,-114.082,-46.112,179.693,4.186,148.770
C05174=1118.745,-114.297,-46.104,179.693,4.182,148.769
C05175=1118.750,-114.512,-46.097,179.693,4.177,148.768
C05176=1118.755,-114.728,-46.089,179.694,4.173,148.767
C05177=1118.760,-114.943,-46.082,179.693,4.168,148.766
C05178=1118.765,-115.193,-46.073,179.694,4.163,148.765
C05179=1118.770,-115.442,-46.064,179.694,4.158,148.764
C05180=1118.776,-115.693,-46.056,179.694,4.153,148.763
C05181=1118.781,-115.943,-46.047,179.694,4.148,148.761
C05182=1118.787,-116.192,-46.039,179.695,4.142,148.760
C05183=1118.792,-116.442,-46.030,179.695,4.137,148.759
C05184=1118.798,-116.692,-46.022,179.695,4.132,148.758
C05185=1118.803,-116.942,-46.013,179.696,4.127,148.756
C05186=1118.808,-117.191,-46.004,179.696,4.121,148.755
C05187=1118.814,-117.441,-45.996,179.696,4.116,148.754
C05188=1118.819,-117.691,-45.987,179.697,4.111,148.753
C05189=1118.824,-117.940,-45.979,179.696,4.105,148.752
C05190=1118.829,-118.190,-45.970,179.697,4.100,148.750
C05191=1118.835,-118.440,-45.962,179.697,4.095,148.749
C05192=1118.841,-118.690,-45.954,179.697,4.090,148.748
C05193=1118.846,-118.939,-45.945,179.698,4.084,148.747
C05194=1118.851,-119.190,-45.937,179.698,4.079,148.745
C05195=1118.857,-119.439,-45.928,179.699,4.074,148.744
C05196=1118.862,-119.690,-45.920,179.699,4.068,148.743
C05197=1118.868,-119.939,-45.911,179.699,4.062,148.742
C05198=1118.873,-120.188,-45.903,179.699,4.057,148.740
C05199=1118.878,-120.439,-45.895,179.699,4.052,148.739
C05200=1118.883,-120.689,-45.886,179.699,4.047,148.738
C05201=1118.889,-120.938,-45.877,179.700,4.042,148.737
C05202=1118.894,-121.188,-45.869,179.701,4.036,148.735
C05203=1118.900,-121.437,-45.861,179.700,4.030,148.734
C05204=1118.905,-121.688,-45.853,179.701,4.025,148.733
C05205=1118.910,-121.937,-45.844,179.701,4.020,148.732
C05206=1118.916,-122.187,-45.836,179.701,4.015,148.730
C05207=1118.921,-122.437,-45.827,179.701,4.010,148.729
C05208=1118.927,-122.687,-45.819,179.702,4.003,148.728
C05209=1118.933,-122.937,-45.811,179.702,3.998,148.727
C05210=1118.937,-123.187,-45.803,179.702,3.993,148.725
C05211=1118.943,-123.436,-45.795,179.703,3.988,148.724
C05212=1118.948,-123.686,-45.786,179.703,3.982,148.723
C05213=1118.954,-123.936,-45.778,179.703,3.976,148.722
C05214=1118.959,-124.186,-45.770,179.703,3.971,148.720
C05215=1118.964,-124.436,-45.761,179.704,3.966,148.719
C05216=1118.970,-124.685,-45.754,179.704,3.961,148.718
C05217=1118.975,-124.935,-45.745,179.704,3.954,148.716
C05218=1118.981,-125.185,-45.738,179.704,3.949,148.715
C05219=1118.986,-125.434,-45.729,179.705,3.944,148.714
C05220=1118.991,-125.685,-45.720,179.705,3.939,148.713
C05221=1118.997,-125.934,-45.712,179.705,3.932,148.711
C05222=1119.002,-126.184,-45.704,179.706,3.927,148.710
C05223=1119.008,-126.434,-45.697,179.706,3.922,148.709
C05224=1119.013,-126.684,-45.688,179.706,3.917,148.708
C05225=1119.019,-126.933,-45.680,179.706,3.910,148.706
C05226=1119.023,-127.148,-45.673,179.706,3.906,148.705
C05227=1119.028,-127.365,-45.666,179.707,3.901,148.704
C05228=1119.032,-127.580,-45.659,179.707,3.896,148.703
C05229=1119.037,-127.795,-45.652,179.707,3.891,148.702
C05230=1119.042,-128.011,-45.645,179.708,3.887,148.701
C05231=1119.047,-128.226,-45.638,179.708,3.882,148.700
C05232=1119.051,-128.442,-45.631,179.708,3.877,148.698
C05233=1119.056,-128.657,-45.624,179.708,3.872,148.697
C05234=1118.633,-128.647,-45.650,179.716,3.876,148.696
C05235=1118.629,-128.432,-45.657,179.715,3.882,148.697
C05236=1118.624,-128.217,-45.664,179.715,3.887,148.698
C05237=1118.619,-128.002,-45.672,179.715,3.891,148.699
C05238=1118.614,-127.786,-45.678,179.714,3.896,148.701
C05239=1118.609,-127.570,-45.685,179.715,3.901,148.702
C05240=1118.604,-127.355,-45.692,179.714,3.905,148.703
C05241=1118.600,-127.140,-45.699,179.714,3.910,148.704
C05242=1118.595,-126.924,-45.706,179.714,3.915,148.705
C05243=1118.590,-126.674,-45.715,179.713,3.920,148.706
C05244=1118.585,-126.424,-45.722,179.713,3.926,148.708
C05245=1118.579,-126.175,-45.731,179.713,3.932,148.709
C05246=1118.574,-125.925,-45.739,179.713,3.937,148.710
C05247=1118.569,-125.676,-45.747,179.712,3.942,148.711
C05248=1118.563,-125.425,-45.755,179.711,3.948,148.713
C05249=1118.558,-125.176,-45.763,179.712,3.954,148.714
C05250=1118.552,-124.926,-45.772,179.711,3.959,148.715
C05251=1118.548,-124.676,-45.780,179.711,3.964,148.716
C05252=1118.542,-124.426,-45.788,179.710,3.970,148.718
C05253=1118.536,-124.176,-45.797,179.711,3.976,148.719
C05254=1118.530,-123.927,-45.804,179.710,3.981,148.720
C05255=1118.525,-123.677,-45.813,179.710,3.986,148.721
C05256=1118.520,-123.427,-45.821,179.710,3.991,148.723
C05257=1118.515,-123.178,-45.830,179.709,3.997,148.724
C05258=1118.509,-122.927,-45.838,179.709,4.003,148.725
C05259=1118.503,-122.678,-45.846,179.709,4.008,148.727
C05260=1118.498,-122.427,-45.854,179.709,4.013,148.728
C05261=1118.494,-122.178,-45.863,179.708,4.018,148.729
C05262=1118.487,-121.928,-45.871,179.708,4.024,148.730
C05263=1118.482,-121.678,-45.879,179.708,4.030,148.732
C05264=1118.477,-121.428,-45.888,179.707,4.035,148.733
C05265=1118.471,-121.179,-45.896,179.707,4.040,148.734
C05266=1118.466,-120.929,-45.905,179.707,4.045,148.735
C05267=1118.460,-120.678,-45.913,179.707,4.050,148.737
C05268=1118.455,-120.430,-45.921,179.706,4.057,148.738
C05269=1118.450,-120.180,-45.930,179.706,4.062,148.739
C05270=1118.445,-119.929,-45.938,179.706,4.067,148.740
C05271=1118.439,-119.680,-45.947,179.706,4.072,148.742
C05272=1118.434,-119.430,-45.956,179.705,4.077,148.743
C05273=1118.428,-119.180,-45.964,179.705,4.083,148.744
C05274=1118.423,-118.931,-45.972,179.705,4.088,148.745
C05275=1118.417,-118.681,-45.981,179.704,4.093,148.747
C05276=1118.412,-118.430,-45.989,179.704,4.099,148.748
C05277=1118.407,-118.181,-45.997,179.704,4.104,148.749
C05278=1118.402,-117.932,-46.006,179.704,4.110,148.750
C05279=1118.397,-117.682,-46.015,179.703,4.115,148.752
C05280=1118.391,-117.432,-46.023,179.703,4.120,148.753
C05281=1118.385,-117.182,-46.032,179.703,4.125,148.754
C05282=1118.380,-116.932,-46.041,179.703,4.130,148.755
C05283=1118.375,-116.682,-46.050,179.702,4.135,148.756
C05284=1118.369,-116.433,-46.058,179.702,4.141,148.758
C05285=1118.364,-116.183,-46.066,179.701,4.146,148.759
C05286=1118.359,-115.933,-46.075,179.701,4.151,148.760
C05287=1118.353,-115.684,-46.084,179.701,4.157,148.761
C05288=1118.347,-115.433,-46.092,179.700,4.162,148.763
C05289=1118.342,-115.183,-46.101,179.701,4.168,148.764
C05290=1118.337,-114.934,-46.110,179.700,4.173,148.765
C05291=1118.332,-114.718,-46.117,179.700,4.177,148.766
C05292=1118.327,-114.503,-46.125,179.700,4.182,148.767
C05293=1118.322,-114.288,-46.132,179.700,4.186,148.768
C05294=1118.318,-114.072,-46.140,179.699,4.190,148.769
C05295=1118.313,-113.857,-46.148,179.699,4.195,148.770
C05296=1118.309,-113.642,-46.155,179.699,4.199,148.771
C05297=1118.304,-113.427,-46.162,179.699,4.204,148.772
C05298=1118.300,-113.211,-46.170,179.698,4.208,148.773
C05299=1118.295,-112.961,-46.178,179.698,4.213,148.775
C05300=1118.289,-112.711,-46.187,179.698,4.219,148.776
C05301=1118.284,-112.462,-46.196,179.697,4.224,148.777
C05302=1118.278,-112.211,-46.205,179.697,4.229,148.778
C05303=1118.273,-111.962,-46.214,179.697,4.234,148.779
C05304=1118.267,-111.712,-46.223,179.697,4.239,148.781
C05305=1118.262,-111.463,-46.232,179.696,4.244,148.782
C05306=1118.257,-111.213,-46.240,179.696,4.250,148.783
C05307=1118.251,-110.963,-46.249,179.696,4.255,148.784
C05308=1118.246,-110.713,-46.258,179.695,4.260,148.785
C05309=1118.241,-110.463,-46.267,179.695,4.265,148.787
C05310=1118.235,-110.214,-46.276,179.695,4.270,148.788
C05311=1118.230,-109.964,-46.285,179.695,4.275,148.789
C05312=1118.224,-109.714,-46.294,179.694,4.281,148.790
C05313=1118.219,-109.464,-46.303,179.694,4.286,148.791
C05314=1118.214,-109.214,-46.312,179.694,4.291,148.793
C05315=1118.209,-108.964,-46.321,179.694,4.296,148.794
C05316=1118.203,-108.715,-46.329,179.693,4.301,148.795
C05317=1118.198,-108.465,-46.338,179.693,4.306,148.796
C05318=1118.193,-108.216,-46.347,179.693,4.312,148.797
C05319=1118.187,-107.965,-46.357,179.692,4.316,148.799
C05320=1118.182,-107.716,-46.366,179.692,4.321,148.800
C05321=1118.176,-107.466,-46.374,179.692,4.326,148.801
C05322=1118.171,-107.216,-46.383,179.691,4.331,148.802
C05323=1118.165,-106.967,-46.392,179.691,4.337,148.803
C05324=1118.160,-106.717,-46.401,179.691,4.342,148.805
C05325=1118.154,-106.467,-46.410,179.691,4.347,148.806
C05326=1118.149,-106.217,-46.419,179.690,4.352,148.807
C05327=1118.144,-105.967,-46.428,179.690,4.357,148.808
C05328=1118.139,-105.717,-46.437,179.690,4.362,148.809
C05329=1118.134,-105.468,-46.447,179.689,4.367,148.811
C05330=1118.128,-105.218,-46.456,179.689,4.372,148.812
C05331=1118.123,-104.968,-46.465,179.689,4.377,148.813
C05332=1118.118,-104.718,-46.474,179.688,4.382,148.814
C05333=1118.113,-104.468,-46.483,179.688,4.387,148.815
C05334=1118.106,-104.219,-46.492,179.688,4.393,148.817
C05335=1118.101,-103.969,-46.501,179.688,4.398,148.818
C05336=1118.096,-103.720,-46.510,179.687,4.402,148.819
C05337=1118.091,-103.470,-46.519,179.687,4.407,148.820
C05338=1118.085,-103.220,-46.529,179.687,4.412,148.821
C05339=1118.080,-102.970,-46.538,179.687,4.417,148.822
C05340=1118.075,-102.720,-46.547,179.687,4.422,148.824
C05341=1118.070,-102.471,-46.556,179.686,4.428,148.825
C05342=1118.064,-102.221,-46.566,179.686,4.433,148.826
C05343=1118.059,-101.971,-46.575,179.685,4.437,148.827
C05344=1118.054,-101.721,-46.583,179.685,4.442,148.828
C05345=1118.048,-101.471,-46.594,179.685,4.447,148.830
C05346=1118.043,-101.222,-46.603,179.685,4.453,148.831
C05347=1118.038,-101.006,-46.610,179.684,4.457,148.832
C05348=1118.034,-100.791,-46.618,179.684,4.461,148.833
C05349=1118.029,-100.576,-46.626,179.684,4.466,148.834
C05350=1118.024,-100.361,-46.634,179.683,4.470,148.835
C05351=1118.020,-100.145,-46.643,179.683,4.474,148.836
C05352=1118.015,-99.930,-46.650,179.682,4.478,148.837
C05353=1118.011,-99.714,-46.658,179.683,4.483,148.838
C05354=1118.006,-99.500,-46.667,179.682,4.487,148.839
C05355=1118.001,-99.250,-46.675,179.682,4.492,148.840
C05356=1117.995,-99.000,-46.685,179.682,4.497,148.841
C05357=1117.990,-98.750,-46.695,179.681,4.501,148.842
C05358=1117.984,-98.500,-46.704,179.681,4.507,148.844
C05359=1117.979,-98.250,-46.713,179.681,4.512,148.845
C05360=1117.974,-98.001,-46.723,179.681,4.517,148.846
C05361=1117.968,-97.751,-46.732,179.680,4.521,148.847
C05362=1117.963,-97.501,-46.741,179.679,4.526,148.848
C05363=1117.957,-97.252,-46.751,179.679,4.532,148.850
C05364=1117.952,-97.002,-46.760,179.679,4.537,148.851
C05365=1117.947,-96.752,-46.769,179.679,4.541,148.852
C05366=1117.942,-96.502,-46.779,179.679,4.546,148.853
C05367=1117.936,-96.252,-46.788,179.678,4.551,148.854
C05368=1117.931,-96.003,-46.798,179.678,4.556,148.855
C05369=1117.926,-95.753,-46.807,179.678,4.561,148.856
C05370=1117.920,-95.503,-46.817,179.677,4.566,148.858
C05371=1117.915,-95.254,-46.826,179.677,4.571,148.859
C05372=1117.910,-95.004,-46.835,179.677,4.576,148.860
C05373=1117.905,-94.754,-46.846,179.676,4.580,148.861
C05374=1117.900,-94.504,-46.855,179.676,4.585,148.862
C05375=1117.894,-94.254,-46.865,179.676,4.591,148.864
C05376=1117.889,-94.004,-46.874,179.675,4.595,148.865
C05377=1117.883,-93.755,-46.884,179.675,4.600,148.866
C05378=1117.878,-93.505,-46.893,179.673,4.605,148.867
C05379=1117.872,-93.255,-46.903,179.673,4.610,148.869
C05380=1117.867,-93.005,-46.912,179.672,4.614,148.870
C05381=1117.862,-92.756,-46.922,179.671,4.619,148.871
C05382=1117.856,-92.506,-46.931,179.671,4.624,148.872
C05383=1117.851,-92.257,-46.941,179.670,4.628,148.873
C05384=1117.846,-92.007,-46.950,179.670,4.634,148.875
C05385=1117.841,-91.756,-46.961,179.669,4.638,148.876
C05386=1117.836,-91.507,-46.970,179.669,4.643,148.877
C05387=1117.830,-91.257,-46.980,179.668,4.648,148.878
C05388=1117.825,-91.007,-46.989,179.668,4.653,148.879
C05389=1117.819,-90.758,-46.999,179.667,4.658,148.881
C05390=1117.814,-90.508,-47.008,179.666,4.663,148.882
C05391=1117.808,-90.258,-47.018,179.666,4.668,148.883
C05392=1117.804,-90.009,-47.028,179.665,4.672,148.884
C05393=1117.798,-89.758,-47.038,179.665,4.677,148.886
C05394=1117.793,-89.509,-47.048,179.665,4.682,148.887
C05395=1117.787,-89.259,-47.057,179.664,4.687,148.888
C05396=1117.782,-89.009,-47.067,179.664,4.692,148.889
C05397=1117.777,-88.759,-47.076,179.663,4.697,148.891
C05398=1117.771,-88.510,-47.086,179.663,4.702,148.892
C05399=1117.766,-88.261,-47.096,179.662,4.707,148.893
C05400=1117.761,-88.010,-47.105,179.662,4.711,148.894
C05401=1117.755,-87.760,-47.116,179.661,4.717,148.896
C05402=1117.750,-87.511,-47.125,179.661,4.722,148.897
C05403=1117.746,-87.296,-47.133,179.660,4.726,148.898
C05404=1117.741,-87.080,-47.142,179.660,4.730,148.899
C05405=1117.736,-86.865,-47.150,179.659,4.734,148.900
C05406=1117.732,-86.650,-47.159,179.659,4.740,148.901
C05407=1117.727,-86.435,-47.167,179.659,4.743,148.902
C05408=1117.723,-86.220,-47.175,179.659,4.747,148.903
C05409=1117.718,-86.004,-47.185,179.658,4.752,148.904
C05410=1117.714,-85.790,-47.193,179.658,4.757,148.905
C05411=1117.708,-85.539,-47.203,179.657,4.761,148.906
C05412=1117.703,-85.290,-47.212,179.657,4.766,148.908
C05413=1117.698,-85.040,-47.223,179.657,4.772,148.909
C05414=1117.693,-84.790,-47.232,179.656,4.777,148.910
C05415=1117.687,-84.541,-47.242,179.656,4.782,148.911
C05416=1117.682,-84.291,-47.252,179.656,4.786,148.912
C05417=1117.677,-84.041,-47.263,179.655,4.791,148.913
C05418=1117.671,-83.791,-47.272,179.655,4.797,148.915
C05419=1117.666,-83.541,-47.282,179.654,4.802,148.916
C05420=1117.660,-83.292,-47.292,179.654,4.807,148.917
C05421=1117.655,-83.043,-47.302,179.654,4.812,148.918
C05422=1117.650,-82.792,-47.311,179.653,4.817,148.920
C05423=1117.644,-82.542,-47.322,179.653,4.822,148.921
C05424=1117.640,-82.293,-47.331,179.653,4.827,148.922
C05425=1117.634,-82.043,-47.341,179.653,4.832,148.923
C05426=1117.629,-81.793,-47.352,179.653,4.837,148.924
C05427=1117.623,-81.544,-47.362,179.653,4.843,148.925
C05428=1117.618,-81.294,-47.371,179.652,4.848,148.927
C05429=1117.613,-81.044,-47.381,179.652,4.853,148.928
C05430=1117.608,-80.794,-47.392,179.652,4.858,148.929
C05431=1117.602,-80.544,-47.402,179.652,4.863,148.930
C05432=1117.597,-80.295,-47.412,179.652,4.868,148.931
C05433=1117.592,-80.046,-47.422,179.651,4.874,148.933
C05434=1117.587,-79.795,-47.432,179.651,4.879,148.934
C05435=1117.581,-79.545,-47.442,179.651,4.884,148.935
C05436=1117.576,-79.296,-47.452,179.651,4.889,148.936
C05437=1117.571,-79.046,-47.462,179.650,4.894,148.937
C05438=1117.565,-78.796,-47.472,179.650,4.900,148.939
C05439=1117.560,-78.547,-47.483,179.650,4.905,148.940
C05440=1117.554,-78.297,-47.493,179.650,4.910,148.941
C05441=1117.550,-78.047,-47.503,179.650,4.915,148.942
C05442=1117.544,-77.798,-47.513,179.650,4.920,148.943
C05443=1117.539,-77.548,-47.523,179.650,4.925,148.944
C05444=1117.534,-77.298,-47.534,179.650,4.930,148.945
C05445=1117.528,-77.048,-47.544,179.650,4.935,148.946
C05446=1117.522,-76.799,-47.554,179.650,4.940,148.948
C05447=1117.517,-76.549,-47.565,179.649,4.946,148.949
C05448=1117.513,-76.299,-47.574,179.649,4.951,148.950
C05449=1117.507,-76.050,-47.585,179.649,4.956,148.951
C05450=1117.502,-75.800,-47.595,179.649,4.962,148.952
C05451=1117.496,-75.550,-47.605,179.649,4.967,148.953
C05452=1117.491,-75.300,-47.616,179.649,4.972,148.955
C05453=1117.486,-75.050,-47.626,179.649,4.977,148.956
C05454=1117.480,-74.801,-47.636,179.649,4.982,148.957
C05455=1117.475,-74.551,-47.647,179.649,4.987,148.958
C05456=1117.470,-74.301,-47.657,179.649,4.992,148.959
C05457=1117.464,-74.051,-47.667,179.649,4.998,148.960
C05458=1117.459,-73.802,-47.677,179.649,5.003,148.961
C05459=1117.454,-73.587,-47.686,179.649,5.007,148.962
C05460=1117.450,-73.371,-47.696,179.650,5.012,148.963
C05461=1117.445,-73.157,-47.704,179.649,5.016,148.964
C05462=1117.441,-72.941,-47.713,179.650,5.021,148.965
C05463=1117.436,-72.726,-47.722,179.650,5.026,148.966
C05464=1117.431,-72.511,-47.731,179.650,5.030,148.967
C05465=1117.427,-72.296,-47.740,179.650,5.035,148.968
C05466=1117.423,-72.081,-47.749,179.650,5.040,148.969
C05467=1117.418,-71.832,-47.760,179.650,5.044,148.970
C05468=1117.413,-71.581,-47.770,179.650,5.049,148.971
C05469=1117.407,-71.332,-47.780,179.650,5.055,148.972
C05470=1117.401,-71.082,-47.791,179.650,5.059,148.973
C05471=1117.396,-70.832,-47.801,179.651,5.065,148.974
C05472=1117.391,-70.583,-47.812,179.651,5.070,148.976
C05473=1117.386,-70.333,-47.823,179.651,5.076,148.977
C05474=1117.381,-70.083,-47.833,179.651,5.080,148.978
C05475=1117.376,-69.833,-47.844,179.651,5.086,148.979
C05476=1117.370,-69.584,-47.854,179.652,5.091,148.980
C05477=1117.365,-69.334,-47.866,179.652,5.096,148.981
C05478=1117.359,-69.084,-47.876,179.652,5.102,148.982
C05479=1117.353,-68.835,-47.886,179.653,5.107,148.983
C05480=1117.349,-68.585,-47.897,179.652,5.112,148.984
C05481=1117.343,-68.335,-47.908,179.653,5.117,148.985
C05482=1117.338,-68.085,-47.918,179.653,5.123,148.986
C05483=1117.333,-67.836,-47.929,179.654,5.128,148.987
C05484=1117.328,-67.586,-47.940,179.654,5.133,148.988
C05485=1117.322,-67.336,-47.950,179.654,5.138,148.989
C05486=1117.317,-67.087,-47.961,179.654,5.143,148.990
C05487=1117.312,-66.837,-47.971,179.655,5.148,148.991
C05488=1117.307,-66.587,-47.982,179.655,5.154,148.992
C05489=1117.301,-66.338,-47.993,179.656,5.159,148.993
C05490=1117.296,-66.087,-48.004,179.655,5.164,148.995
C05491=1117.290,-65.838,-48.014,179.656,5.170,148.996
C05492=1117.286,-65.588,-48.025,179.657,5.174,148.996
